# B&R Automation Studio project VisionSample (part 4)

#### Main.st - Init, cyclic, exit code
```iecst
// --------------------------------------------------------------------------------------------------------------------
// Vision image upload task. This task stores the camera image on the file device media
// Version 2.0
// --------------------------------------------------------------------------------------------------------------------
PROGRAM _INIT
	gVisionImage.CFG.FileDevice 	:= 'VisionFileDevice';		// File device name where the images are stored
	gVisionImage.CFG.DirName		:= 'Vision';				// Directory used for images

	gVisionImage.CMD.CreateDir	:= TRUE;
	gVisionImage.DAT.ImageSelected	:= '';

	brsmemcpy(ADR(b64key), ADR('ABCDEFGHIJKLMNOPQRSTUVWXYZabcdefghijklmnopqrstuvwxyz0123456789+/'), SIZEOF(b64key));

	// Create memory for uploading and transforming image
	// Size: a 5MP picture in bmp format has less than 6.000.000 Bytes. A SVG with bas64 conversion maximum the 4/3 size.
	MemUploadSize		:= 6000000;
	MemSvgHeaderSize	:= 2000;
	MemSvgCrosshSize	:= 18000;
	MemSvgSize			:= MemUploadSize * 4 / 3 + MemSvgHeaderSize + MemSvgCrosshSize;
	AsMemPartCreate_0.enable	:= TRUE;
	AsMemPartCreate_0.len		:= MemUploadSize + MemSvgSize + MemSvgCrosshSize + 1000; // 1000 Bytes for AsMemPart stuff/header
	AsMemPartCreate_0();

	IF AsMemPartCreate_0.status = 0 THEN
		AsMemPartAllocClear_0.enable	:= TRUE;
		AsMemPartAllocClear_0.ident		:= AsMemPartCreate_0.ident;
		AsMemPartAllocClear_0.len		:= MemUploadSize;
		AsMemPartAllocClear_0();
		IF AsMemPartAllocClear_0.status = 0 THEN
			MemUpload := AsMemPartAllocClear_0.mem;
		END_IF
		AsMemPartAllocClear_0.len		:= MemSvgSize;
		AsMemPartAllocClear_0();
		IF AsMemPartAllocClear_0.status = 0 THEN
			MemSvg := AsMemPartAllocClear_0.mem;
		END_IF
		AsMemPartAllocClear_0.len		:= MemSvgCrosshSize;
		AsMemPartAllocClear_0();
		IF AsMemPartAllocClear_0.status = 0 THEN
			MemSvgCrossh := AsMemPartAllocClear_0.mem;
		END_IF
	END_IF
	ACTION_InitTexts;
END_PROGRAM

// -----------------------------------------------------------------------------------------------------------
// Cyclic part
// -----------------------------------------------------------------------------------------------------------
PROGRAM _CYCLIC

	// -----------------------------------------------------------------------------------------------------------
	// State machine for uploading the image
	// -----------------------------------------------------------------------------------------------------------
	CASE Step OF
		// -----------------------------------------------------------------------------------------------------------
		// Wait for new upload command
		VISTEP_WAIT:
			gVisionImage.DAT.Status := 0;

			// -----------------------------------------------------------------------------------------------------------
			// Create the internal directory VisionImageArchive
			IF gVisionImage.CMD.CreateDir THEN
				gVisionImage.DAT.Status := 65535;
				Step := VISTEP_CREATE_DIR;

			// -----------------------------------------------------------------------------------------------------------
			// Delete image directory
			ELSIF gVisionImage.CMD.DeleteDir THEN
				gVisionImage.DAT.Status := 65535;
				Step := VISTEP_DELETE_DIR;

			// -----------------------------------------------------------------------------------------------------------
			// Refresh image data from file device
			ELSIF gVisionImage.CMD.Refresh THEN
				gVisionImage.DAT.Status := 65535;
				Step := VISTEP_READ_DIR1;

			// -----------------------------------------------------------------------------------------------------------
			// Delete image data from file device
			ELSIF gVisionImage.CMD.DeleteImage THEN
				IF brsstrlen(ADR(gVisionImage.DAT.ImageSelected)) > 0 THEN
					brsstrcpy(ADR(FileNamePict), ADR(gVisionImage.CFG.DirName));
					brsstrcat(ADR(FileNamePict), ADR('/'));
					brsstrcat(ADR(FileNamePict), ADR(gVisionImage.DAT.ImageSelected));
					gVisionImage.DAT.Status := 65535;
					Step := VISTEP_DELETE_IMAGE;
				ELSE
					gVisionImage.CMD.DeleteImage := FALSE;
				END_IF

				// -----------------------------------------------------------------------------------------------------------
				// Save image from camera
			ELSIF gVisionImage.CMD.GetImage THEN
				FileNamePict := gVisionImage.CFG.DirName;
				brsstrcat(ADR(FileNamePict), ADR('/last_image.bmp'));

				ViBaseGetImage_0.Execute := FALSE;
				ViBaseGetImage_0();

				gVisionImage.DAT.Status		:= 65535;
				Step						:= VISTEP_DELETE_IMAGE;

				// -----------------------------------------------------------------------------------------------------------
				// Save image from camera
			ELSIF gVisionImage.CMD.SaveImage THEN
				// Generate file name if not provided
				IF gVisionImage.CFG.FileName = '' THEN
					// Generate new file name
					DTGetTime_0.enable := 1;
					DTGetTime_0();
					DT_TO_DTStructure(DTGetTime_0.DT1, ADR(DTStructure_0));
					FileNamePict := gVisionImage.CFG.DirName;
					brsstrcat(ADR(FileNamePict), ADR('/'));
					tmpStr1 := UINT_TO_STRING(DTStructure_0.year);
					brsstrcat(ADR(FileNamePict), ADR(tmpStr1));
					brsstrcat(ADR(FileNamePict), ADR('_'));
					tmpStr1 := USINT_TO_STRING(DTStructure_0.month);
					IF(DTStructure_0.month < 10) THEN
						brsstrcat(ADR(FileNamePict), ADR('0'));
					END_IF
					brsstrcat(ADR(FileNamePict), ADR(tmpStr1));
					brsstrcat(ADR(FileNamePict), ADR('_'));
					tmpStr1 := USINT_TO_STRING(DTStructure_0.day);
					IF(DTStructure_0.day < 10) THEN
						brsstrcat(ADR(FileNamePict), ADR('0'));
					END_IF
					brsstrcat(ADR(FileNamePict), ADR(tmpStr1));
					brsstrcat(ADR(FileNamePict), ADR('_'));
					tmpStr1 := USINT_TO_STRING(DTStructure_0.hour);
					IF(DTStructure_0.hour < 10) THEN
						brsstrcat(ADR(FileNamePict), ADR('0'));
					END_IF
					brsstrcat(ADR(FileNamePict), ADR(tmpStr1));
					brsstrcat(ADR(FileNamePict), ADR('_'));
					tmpStr1 := USINT_TO_STRING(DTStructure_0.minute);
					IF(DTStructure_0.minute < 10) THEN
						brsstrcat(ADR(FileNamePict), ADR('0'));
					END_IF
					brsstrcat(ADR(FileNamePict), ADR(tmpStr1));
					brsstrcat(ADR(FileNamePict), ADR('_'));
					tmpStr1 := USINT_TO_STRING(DTStructure_0.second);
					IF(DTStructure_0.second < 10) THEN
						brsstrcat(ADR(FileNamePict), ADR('0'));
					END_IF
					brsstrcat(ADR(FileNamePict), ADR(tmpStr1));
				ELSE
					FileNamePict := gVisionImage.CFG.FileName;
				END_IF

				brsstrcpy(ADR(FileNameSvg), ADR(FileNamePict));
				brsstrcat(ADR(FileNameSvg), ADR('.svg'));
				brsstrcat(ADR(FileNamePict), ADR('.bmp'));

				ViBaseGetImage_0.Execute := FALSE;
				ViBaseGetImage_0();

				gVisionImage.DAT.Status		:= 65535;
				Step						:= VISTEP_DELETE_IMAGE;

			// -----------------------------------------------------------------------------------------------------------
			// Reset error
			ELSIF gVisionImage.CMD.ResetError THEN
				gVisionImage.CMD.ResetError := FALSE;
			END_IF

			// -----------------------------------------------------------------------------------------------------------
			// Load new image into window
			IF visImageSelectedOld <> gVisionImage.DAT.ImageSelected AND dir_entry > 0 THEN
				brsmemset(ADR(gVisionImage.DAT.ImagePath), 0, SIZEOF(gVisionImage.DAT.ImagePath));
				brsmemset(ADR(tmpStr1), 0, SIZEOF(tmpStr1));
				gVisionImage.DAT.ImagePath := '/FileDevice:';
				brsstrcat(ADR(gVisionImage.DAT.ImagePath), ADR(gVisionImage.CFG.FileDevice));
				brsstrcat(ADR(gVisionImage.DAT.ImagePath), ADR('/'));
				brsstrcat(ADR(gVisionImage.DAT.ImagePath), ADR(gVisionImage.CFG.DirName));
				brsstrcat(ADR(gVisionImage.DAT.ImagePath), ADR('/'));
				brsstrcat(ADR(gVisionImage.DAT.ImagePath), ADR(gVisionImage.DAT.ImageSelected));
			END_IF
			visImageSelectedOld := gVisionImage.DAT.ImageSelected;

		// -----------------------------------------------------------------------------------------------------------
		// Create directory on User-Partition, if not exists
		// -----------------------------------------------------------------------------------------------------------
		VISTEP_CREATE_DIR:
			DirCreate_0.enable	:= TRUE;
			DirCreate_0.pDevice	:= ADR(gVisionImage.CFG.FileDevice);
			DirCreate_0.pName	:= ADR(gVisionImage.CFG.DirName);
			DirCreate_0();

			IF DirCreate_0.status = 0 OR DirCreate_0.status = fiERR_DIR_ALREADY_EXIST THEN
				Step := VISTEP_READ_DIR1;
			ELSIF DirCreate_0.status <> 65535 THEN
				gVisionImage.DAT.Status := DirCreate_0.status;
				Step := VISTEP_ERR;
			END_IF

		// -----------------------------------------------------------------------------------------------------------
		// Delete directory on User-Partition
		// -----------------------------------------------------------------------------------------------------------
		VISTEP_DELETE_DIR:
			DirDeleteEx_0.enable	:= TRUE;
			DirDeleteEx_0.pDevice	:= ADR(gVisionImage.CFG.FileDevice);
			DirDeleteEx_0.pName		:= ADR(gVisionImage.CFG.DirName);
			DirDeleteEx_0();

			IF DirDeleteEx_0.status = 0 THEN
				Step := VISTEP_CREATE_DIR;
			ELSIF DirDeleteEx_0.status <> 65535 THEN
				gVisionImage.DAT.Status := DirDeleteEx_0.status;
				Step := VISTEP_ERR;
			END_IF

		// -----------------------------------------------------------------------------------------------------------
		// Read all existing image names from directory
		// -----------------------------------------------------------------------------------------------------------
		VISTEP_READ_DIR1:
			// Clear all memory
			brsmemset(ADR(gVisionImage.DAT.ImagesList), 0, SIZEOF(gVisionImage.DAT.ImagesList));
			brsmemset(ADR(gVisionImage.DAT.ImageSelected), 0, SIZEOF(gVisionImage.DAT.ImageSelected));
			visImageSelectedOld := '';
			gVisionImage.DAT.ImageSelected	:= '';
			dir_entry			:= 0;
			idx					:= 0;
			file_newest			:= '';
			file_oldest			:= '';
			date_newest			:= UDINT_TO_DT(0);
			date_oldest			:= DT#2100-06-06-12:00:00;
			cmdDeleteOldest		:= FALSE;
			Step := VISTEP_READ_DIR2;

		// -----------------------------------------------------------------------------------------------------------
		// Proceed with next entry
		// -----------------------------------------------------------------------------------------------------------
		VISTEP_READ_DIR2:
			DirRead_0.enable 	:= 1;
			DirRead_0.pDevice 	:= ADR(gVisionImage.CFG.FileDevice);
			DirRead_0.pPath		:= ADR(gVisionImage.CFG.DirName);
			DirRead_0.entry 	:= idx;
			DirRead_0.option 	:= fiFILE;
			DirRead_0.pData 	:= ADR(dir_data);
			DirRead_0.data_len 	:= SIZEOF(dir_data);
			DirRead_0();

			IF DirRead_0.status = 0 THEN
				// Make sure file is an image and we have space to store them
				IF  brsstrcmp(ADR(dir_data.Filename) + brsstrlen(ADR(dir_data.Filename)) - 4, ADR('.bmp')) = 0 OR
					brsstrcmp(ADR(dir_data.Filename) + brsstrlen(ADR(dir_data.Filename)) - 4, ADR('.jpg')) = 0 OR
					brsstrcmp(ADR(dir_data.Filename) + brsstrlen(ADR(dir_data.Filename)) - 4, ADR('.svg')) = 0 THEN
					// Find newest and oldest file
					IF dir_data.Date > date_newest THEN
						brsstrcpy(ADR(file_newest), ADR(dir_data.Filename));
						date_newest := dir_data.Date;
					END_IF
					IF dir_data.Date < date_oldest THEN
						brsstrcpy(ADR(file_oldest), ADR(dir_data.Filename));
						date_oldest := dir_data.Date;
					END_IF
					IF dir_entry <= SIZEOF(gVisionImage.DAT.ImagesList)/SIZEOF(gVisionImage.DAT.ImagesList[0]) - 1 THEN
						// Create list box data
						gVisionImage.DAT.ImagesList[dir_entry] := '{"value":"';
						brsstrcat(ADR(gVisionImage.DAT.ImagesList[dir_entry]), ADR(dir_data.Filename));
						brsstrcat(ADR(gVisionImage.DAT.ImagesList[dir_entry]), ADR('","text":"'));
						brsstrcat(ADR(gVisionImage.DAT.ImagesList[dir_entry]), ADR(dir_data.Filename));
						brsstrcat(ADR(gVisionImage.DAT.ImagesList[dir_entry]), ADR('"}'));
						dir_entry := dir_entry + 1;
					ELSE
						cmdDeleteOldest := TRUE;
					END_IF
				END_IF
				idx := idx + 1;
			ELSIF DirRead_0.status = fiERR_NO_MORE_ENTRIES THEN
				IF cmdDeleteOldest THEN
					brsstrcpy(ADR(tmpStr1), ADR(gVisionImage.CFG.DirName));
					brsstrcat(ADR(tmpStr1), ADR('/'));
					brsstrcat(ADR(tmpStr1), ADR(file_oldest));
					Step := VISTEP_DELETE_IMAGE;
				ELSE
					TON_VisPause(IN := FALSE);
					Step := VISTEP_READ_DIR3;
				END_IF
			ELSIF DirRead_0.status <> 65535 THEN
				gVisionImage.DAT.Status := DirRead_0.status;
				Step := VISTEP_ERR;
			END_IF

		// -----------------------------------------------------------------------------------------------------------
		// Wait for vis before setting last file
		// -----------------------------------------------------------------------------------------------------------
		VISTEP_READ_DIR3:
			TON_VisPause.IN := TRUE;
			TON_VisPause.PT := T#250ms;
			TON_VisPause();

			IF TON_VisPause.Q THEN
				brsstrcpy(ADR(gVisionImage.DAT.ImageSelected), ADR(file_newest));
				brsmemset(ADR(gVisionImage.CMD), 0, SIZEOF(gVisionImage.CMD));
				Step := VISTEP_WAIT;
			END_IF

		// -----------------------------------------------------------------------------------------------------------
		// Delete Image
		// -----------------------------------------------------------------------------------------------------------
		VISTEP_DELETE_IMAGE:
			cmdDeleteOldest			:= FALSE;
			FileDelete_0.enable 	:= 1;
			FileDelete_0.pDevice	:= ADR(gVisionImage.CFG.FileDevice);
			FileDelete_0.pName 		:= ADR(FileNamePict);
			FileDelete_0();

			IF (FileDelete_0.status = 0 OR FileDelete_0.status = fiERR_FILE_NOT_FOUND) AND (gVisionImage.CMD.GetImage OR gVisionImage.CMD.SaveImage) THEN
				Step := VISTEP_REQUEST;
			ELSIF FileDelete_0.status = 0 THEN
				Step := VISTEP_READ_DIR1;
			ELSIF FileDelete_0.status <> 65535 THEN
				gVisionImage.DAT.Status := FileDelete_0.status;
				Step := VISTEP_ERR;
			END_IF

		// -----------------------------------------------------------------------------------------------------------
		// Get new image
		// -----------------------------------------------------------------------------------------------------------
		VISTEP_REQUEST:
			ViBaseGetImage_0.MpLink := ADR(gVisionImage.CFG.ComponentLink);
			ViBaseGetImage_0.Execute := TRUE;
			ViBaseGetImage_0.Type :=  viBASE_IMAGE_TYPE_BMP;
			//ViBaseGetImage_0.QualityLevel := ;
			ViBaseGetImage_0.Timeout := T#10s;
			ViBaseGetImage_0.Buffer := MemUpload;
			ViBaseGetImage_0.BufferSize := MemUploadSize;
			ViBaseGetImage_0();

			IF ViBaseGetImage_0.Busy = 0 THEN
				IF ViBaseGetImage_0.StatusID = 0 THEN
					Step := VISTEP_SAVE1;
				ELSIF ViBaseGetImage_0.StatusID <> ERR_FUB_BUSY THEN
					gVisionImage.DAT.Status := ViBaseGetImage_0.StatusID;
					Step := VISTEP_ERR;
				END_IF
			END_IF

		// -----------------------------------------------------------------------------------------------------------
		// Save image
		// -----------------------------------------------------------------------------------------------------------
		VISTEP_SAVE1:
			FileCreate_0.enable		:= TRUE;
			FileCreate_0.pDevice	:= ADR(gVisionImage.CFG.FileDevice);
			FileCreate_0.pFile		:= ADR(FileNamePict);
			FileCreate_0();

			IF FileCreate_0.status = 0 THEN
				Step := VISTEP_SAVE2;
			ELSIF FileCreate_0.status <> ERR_FUB_BUSY THEN
				gVisionImage.DAT.Status := FileCreate_0.status;
				Step := VISTEP_ERR;
			END_IF

		VISTEP_SAVE2:
			FileWrite_0.enable		:= TRUE;
			FileWrite_0.ident		:= FileCreate_0.ident;
			FileWrite_0.offset		:= 0;
			FileWrite_0.pSrc		:= MemUpload;
			FileWrite_0.len			:= ViBaseGetImage_0.BufferLen;
			FileWrite_0();

			IF FileWrite_0.status = 0 THEN
				Step := VISTEP_SAVE3;
			ELSIF FileWrite_0.status <> ERR_FUB_BUSY THEN
				gVisionImage.DAT.Status := FileWrite_0.status;
				Step := VISTEP_ERR;
			END_IF

		VISTEP_SAVE3:
			FileClose_0.enable		:= TRUE;
			FileClose_0.ident		:= FileCreate_0.ident;
			FileClose_0();

			IF FileClose_0.status = 0 THEN
				image_idx := image_idx + 1;
				brsitoa(image_idx, ADR(tmpStr1));
				gVisionImage.DAT.ImageLast := '/FileDevice:';
				brsstrcat(ADR(gVisionImage.DAT.ImageLast), ADR(gVisionImage.CFG.FileDevice));
				brsstrcat(ADR(gVisionImage.DAT.ImageLast), ADR('/'));
				brsstrcat(ADR(gVisionImage.DAT.ImageLast), ADR(gVisionImage.CFG.DirName));
				brsstrcat(ADR(gVisionImage.DAT.ImageLast), ADR('/last_image.bmp?'));
				brsstrcat(ADR(gVisionImage.DAT.ImageLast), ADR(tmpStr1));

				IF gVisionImage.CMD.SaveImage THEN
					Step := VISTEP_SVG_PREPARE;
				ELSE
					gVisionImage.CMD.GetImage := FALSE;
					Step := VISTEP_WAIT;
				END_IF
			ELSIF FileClose_0.status <> ERR_FUB_BUSY THEN
				gVisionImage.DAT.Status := FileClose_0.status;
				Step := VISTEP_ERR;
			END_IF

		// -----------------------------------------------------------------------------------------------------------
		// Create SVG file with image and crosshair/texts
		// -----------------------------------------------------------------------------------------------------------
		VISTEP_SVG_PREPARE:
			b64neededOutput	:= (ViBaseGetImage_0.BufferLen/3)*4 + BOOL_TO_UDINT(UDINT_TO_BOOL(ViBaseGetImage_0.BufferLen MOD 3))*4;
			IF b64neededOutput < MemSvgSize - MemSvgHeaderSize - MemSvgCrosshSize THEN
				brsmemset(MemSvg, 0, MemSvgSize); // clear complete memory
				// Prepare the svg header up to the base64 picture data
				brsstrcpy(MemSvg, ADR(SvgTexts.Header1));
				brsstrcat(MemSvg, ADR(FileNameSvg));
				brsstrcat(MemSvg, ADR(SvgTexts.Header2));
				brsstrcat(MemSvg, ADR('bmp'));
				brsstrcat(MemSvg, ADR(SvgTexts.Header3));
				Step := VISTEP_SVG_BAS64_1;
			ELSE
				gVisionImage.DAT.Status := ERR_BUFF_TOO_SMALL;
				Step := VISTEP_ERR;
			END_IF

		// -----------------------------------------------------------------------------------------------------------
		// Code picture data with Base64 to embedd the picture into a svg file
		VISTEP_SVG_BAS64_1:
			b64AdrInBuffer	:= MemUpload; 						// Original bmp or jpg picture
			b64AdrOutBuffer	:= MemSvg + brsstrlen(MemSvg); 		// Write to the end of the actual svg data
			b64actposIN		:= b64AdrInBuffer;
			b64actposOUT	:= b64AdrOutBuffer;
			Step := VISTEP_SVG_BAS64_2;

		VISTEP_SVG_BAS64_2:
			FOR i := 0 TO CONVERT_CYCLES DO
				IF b64actposIN < b64AdrInBuffer + ViBaseGetImage_0.BufferLen THEN
					b64blockLen := UDINT_TO_USINT(LIMIT(0, b64AdrInBuffer + ViBaseGetImage_0.BufferLen - b64actposIN, 3));
					b64in ACCESS b64actposIN;
					b64out ACCESS b64actposOUT;
					b64out[0]		:= b64key[ SHR(b64in[0],2) ];
					IF b64blockLen = 1 THEN
						b64out[1]	:= b64key[ SHL((b64in[0] AND 16#03),4)];
						b64out[2]	:= 61;
						b64out[3]	:= 61;
					ELSIF b64blockLen = 2 THEN
						b64out[1]	:= b64key[ SHL((b64in[0] AND 16#03),4) OR SHR(b64in[1],4) ];
						b64out[2]	:= b64key[ SHL((b64in[1] AND 16#0F),2)];
						b64out[3]	:= 61;
					ELSIF b64blockLen = 3 THEN
						b64out[1]	:= b64key[ SHL((b64in[0] AND 16#03),4) OR SHR(b64in[1],4) ];
						b64out[2]	:= b64key[ SHL((b64in[1] AND 16#0F),2) OR SHR(b64in[2],6) ];
						b64out[3]	:= b64key[ b64in[2] AND 16#3F ];
					END_IF
					b64actposIN		:= b64actposIN + 3;
					b64actposOUT	:= b64actposOUT + 4;
				ELSE
					Step := VISTEP_SVG_CROSSH;
					EXIT;
				END_IF

			END_FOR

		// -----------------------------------------------------------------------------------------------------------
		// Prepare the second part after base64 picture data
		VISTEP_SVG_CROSSH:
			brsmemset(MemSvgCrossh, 0, MemSvgCrosshSize);
			brsstrcat(MemSvgCrossh, ADR(SvgTexts.Header4));
			brsstrcat(MemSvgCrossh, ADR(SvgTexts.CrosshairDefinition));
			FOR i := 1 TO MAX_NUM_RESULTS DO
				IF gVisionImage.DAT.Crosshair[i].CrosshairX <> 0 AND gVisionImage.DAT.Crosshair[i].CrosshairY <> 0 THEN
					brsstrcat(MemSvgCrossh, ADR(SvgTexts.Crosshair1));
					brsitoa(REAL_TO_DINT(gVisionImage.DAT.Crosshair[i].CrosshairX), ADR(tmpStr1));
					brsstrcat(MemSvgCrossh, ADR(tmpStr1));
					brsstrcat(MemSvgCrossh, ADR(','));
					brsitoa(REAL_TO_DINT(gVisionImage.DAT.Crosshair[i].CrosshairY), ADR(tmpStr1));
					brsstrcat(MemSvgCrossh, ADR(tmpStr1));
					brsstrcat(MemSvgCrossh, ADR(') rotate('));
					brsitoa(REAL_TO_DINT(gVisionImage.DAT.Crosshair[i].CrosshairRotate), ADR(tmpStr1));
					brsstrcat(MemSvgCrossh, ADR(tmpStr1));
					brsstrcat(MemSvgCrossh, ADR(',40,40)"/>'));
				END_IF
			END_FOR
			FOR i := 1 TO MAX_NUM_RESULTS DO
				IF gVisionImage.DAT.Crosshair[i].CrosshairX <> 0 AND gVisionImage.DAT.Crosshair[i].CrosshairY <> 0 THEN
					brsstrcat(MemSvgCrossh, ADR('$r$n$t'));
					brsstrcat(MemSvgCrossh, ADR(gVisionImage.DAT.Crosshair[i].Text));
				END_IF
			END_FOR
			brsstrcat(MemSvgCrossh, ADR(SvgTexts.SvgClose));
			Step := VISTEP_SVG_CONCAT;

		VISTEP_SVG_CONCAT:
			brsstrcat(MemSvg, MemSvgCrossh);
			Step := VISTEP_SVG_SAVE1;

		// -----------------------------------------------------------------------------------------------------------
		// Save SVG file
		// -----------------------------------------------------------------------------------------------------------
		VISTEP_SVG_SAVE1:
			FileCreate_0.enable		:= TRUE;
			FileCreate_0.pDevice	:= ADR(gVisionImage.CFG.FileDevice);
			FileCreate_0.pFile		:= ADR(FileNameSvg);
			FileCreate_0();

			IF FileCreate_0.status = 0 THEN
				Step := VISTEP_SVG_SAVE2;
			ELSIF FileCreate_0.status <> ERR_FUB_BUSY THEN
				gVisionImage.DAT.Status := FileCreate_0.status;
				Step := VISTEP_ERR;
			END_IF

		VISTEP_SVG_SAVE2:
			FileWrite_0.enable		:= TRUE;
			FileWrite_0.ident		:= FileCreate_0.ident;
			FileWrite_0.offset		:= 0;
			FileWrite_0.pSrc		:= MemSvg;
			FileWrite_0.len			:= brsstrlen(MemSvg);
			FileWrite_0();

			IF FileWrite_0.status = 0 THEN
				Step := VISTEP_SVG_SAVE3;
			ELSIF FileWrite_0.status <> ERR_FUB_BUSY THEN
				gVisionImage.DAT.Status := FileWrite_0.status;
				Step := VISTEP_ERR;
			END_IF

		VISTEP_SVG_SAVE3:
			FileClose_0.enable		:= TRUE;
			FileClose_0.ident		:= FileCreate_0.ident;
			FileClose_0();

			IF FileClose_0.status = 0 THEN
				Step := VISTEP_READ_DIR1;
			ELSIF FileClose_0.status <> ERR_FUB_BUSY THEN
				gVisionImage.DAT.Status := FileClose_0.status;
				Step := VISTEP_ERR;
			END_IF

		// -----------------------------------------------------------------------------------------------------------
		// Error state
		// -----------------------------------------------------------------------------------------------------------
		VISTEP_ERR:
			// Reset all commands and wait or ack
			ViBaseGetImage_0.Execute	:= TRUE;
			ViBaseGetImage_0();

			IF gVisionImage.CMD.ResetError THEN
				gVisionImage.CMD.ResetError := FALSE;
				Step := VISTEP_WAIT;
			END_IF
			brsmemset(ADR(gVisionImage.CMD), 0, SIZEOF(gVisionImage.CMD));
	END_CASE

END_PROGRAM
```

#### Types.typ - Local data types
```iecst
TYPE
	VIStep_Enum :
		(
		VISTEP_WAIT,
		VISTEP_GEN_CROSSHAIR,
		VISTEP_CREATE_DIR,
		VISTEP_DELETE_DIR,
		VISTEP_READ_DIR1,
		VISTEP_READ_DIR2,
		VISTEP_READ_DIR3,
		VISTEP_DELETE_IMAGE,
		VISTEP_REQUEST1,
		VISTEP_REQUEST2,
		VISTEP_REQUEST3,
		VISTEP_SAVE1,
		VISTEP_SAVE2,
		VISTEP_SAVE3,
		VISTEP_SVG_CROSSH,
		VISTEP_SVG_CONCAT,
		VISTEP_ERR
		);
	SvgTexts_Type : 	STRUCT
		Header1 : STRING[500];
		Header2 : STRING[500];
		Header3 : STRING[500];
		Header4 : STRING[500];
		CrosshairDefinition : STRING[1000];
		Crosshair1 : STRING[500];
		SvgClose : STRING[50];
	END_STRUCT;
	DiagTime_Type : 	STRUCT
		Refresh : TIME;
		BeginSaveBMPJPG : TIME;
		EndSaveBMPJPG : TIME;
		BeginSVG : TIME;
		BeginSVGSave : TIME;
		EndSVGSave : TIME;
	END_STRUCT;
END_TYPE
```

#### Variables.var - Local variables
```iecst
VAR
	Step : VIStep_Enum;
	tmpStr1 : STRING[80];
	idx : UINT;
END_VAR
(**)
(*Filehandling*)
VAR
	DirCreate_0 : DirCreate;
	DirDeleteEx_0 : DirDeleteEx;
	FileNamePict : STRING[80];
	FileNameSvg : STRING[80];
	FileCreate_0 : FileCreate;
	FileDelete_0 : FileDelete;
	FileWrite_0 : FileWrite;
	FileClose_0 : FileClose;
	DirRead_0 : DirRead;
	dir_data : fiDIR_READ_DATA;
	dir_entry : UINT;
	file_newest : STRING[80];
	file_oldest : STRING[80];
	date_newest : DATE_AND_TIME;
	date_oldest : DATE_AND_TIME;
	cmdDeleteOldest : BOOL;
	image_idx : UINT;
	DTGetTime_0 : DTGetTime;
	DTStructure_0 : DTStructure;
	TON_VisPause : TON;
END_VAR
(**)
(*mappView connected variables*)
VAR
	visImageSelectedOld : STRING[80];
END_VAR
(**)
(*Create memory*)
VAR
	AsMemPartCreate_0 : AsMemPartCreate;
	AsMemPartAllocClear_0 : AsMemPartAllocClear;
	MemUpload : UDINT;
	MemUploadSize : UDINT;
	MemSvg : UDINT;
	MemSvgSize : UDINT;
	MemSvgHeaderSize : UDINT;
	MemSvgCrossh : UDINT;
	MemSvgCrosshSize : UDINT;
END_VAR
(**)
VAR
	ViBaseGetImage_0 : ViBaseGetImage;
END_VAR
(**)
(*Bas64*)
VAR
	b64AdrInBuffer : UDINT;
	b64AdrOutBuffer : UDINT;
	b64neededOutput : UDINT;
	b64key : ARRAY[0..63] OF USINT;
	b64actposIN : UDINT;
	b64actposOUT : UDINT;
	b64in : REFERENCE TO ARRAY[0..2] OF USINT;
	b64out : REFERENCE TO ARRAY[0..3] OF USINT;
	b64blockLen : USINT;
	SvgTexts : SvgTexts_Type;
	i : UDINT;
END_VAR
(**)
(*Constants*)
VAR
	ERR_BUFF_TOO_SMALL : UINT := 50001;
END_VAR
```

#### LocalFunctions.fun - not listed in the package file held
```iecst
FUNCTION_BLOCK ViDownloadImage (* *) (*$GROUP=User,$CAT=User,$GROUPICON=User.png,$CATICON=User.png*)
	VAR_INPUT
		Enable : BOOL;
		FileDevice : STRING[80];
		FileName : STRING[80];
		ImgName : STRING[80];
		visDownloadFileUrl : REFERENCE TO STRING[200];
	END_VAR
	VAR_OUTPUT
		Status : UINT;
	END_VAR
	VAR
		Step : INT;
		AsMemPartCreate_0 : AsMemPartCreate;
		AsMemPartAllocClear_0 : AsMemPartAllocClear;
		MemSvgAdr : UDINT;
		MemSvgSize : UDINT;
		FileOpen_0 : FileOpen;
		FileRead_0 : FileRead;
		FileClose_0 : FileClose;
		TON_Timeout : TON;
		httpService_Download : httpService;
		response_header : httpResponseHeader_t;
		response_header_data : STRING[300];
	END_VAR
END_FUNCTION_BLOCK

FUNCTION_BLOCK ViRefreshImageList
	VAR_INPUT
		Enable : BOOL;
		VisionImage : REFERENCE TO typVisionImage;
		ImageList : REFERENCE TO ARRAY[0..19] OF STRING[80];
		visSelectedImage : REFERENCE TO STRING[80];
	END_VAR
	VAR_OUTPUT
		Status : UINT;
		DirEntries : UINT;
	END_VAR
	VAR
		Step : INT;
		visSelectedImageOld : STRING[80];
		idx : UINT;
		file_newest : STRING[80];
		file_oldest : STRING[80];
		date_newest : DATE_AND_TIME;
		date_oldest : DATE_AND_TIME;
		cmdDeleteOldest : BOOL;
		DirRead_0 : DirRead;
		FileDelete_0 : FileDelete;
		dir_data : fiDIR_READ_DATA;
		DeleteFileName : STRING[80];
		TON_VisPause : TON;
	END_VAR
END_FUNCTION_BLOCK

FUNCTION_BLOCK ViSaveImgOnPlc
	VAR_INPUT
		Enable : BOOL;
		CFG : typVisionImageConfig;
		PowerlinkNode : USINT;
		CrossHairInfo : REFERENCE TO ARRAY[0..MAX_NUM_RESULTS] OF typCrossHairInfo;
	END_VAR
	VAR_OUTPUT
		Status : UINT;
	END_VAR
	VAR
		Step : INT;
		AsMemPartCreate_0 : AsMemPartCreate;
		AsMemPartAllocClear_0 : AsMemPartAllocClear;
		MemInfo : MemInfoSave_Type;
		DiagStartTime : TIME;
		DiagTime : DiagTime_Type;
		DTGetTime_0 : DTGetTime;
		DTStructure_0 : DTStructure;
		FileNameImg : STRING[80];
		FileNameSvg : STRING[80];
		URI : STRING[80];
		Host : STRING[80];
		httpClient_0 : httpClient;
		httpClientErrorStatus : UINT;
		RequestHeader : httpRequestHeader_t;
		TON_ReloadTimeout : TON;
		UploadedImgSize : UDINT;
		FileCreate_0 : FileCreate;
		FileWrite_0 : FileWrite;
		FileClose_0 : FileClose;
		b64AdrInBuffer : UDINT;
		b64AdrOutBuffer : UDINT;
		b64neededOutput : UDINT;
		b64key : ARRAY[0..63] OF USINT;
		b64actposIN : UDINT;
		b64actposOUT : UDINT;
		b64in : REFERENCE TO ARRAY[0..2] OF USINT;
		b64out : REFERENCE TO ARRAY[0..3] OF USINT;
		b64blockLen : UINT;
		FirstElement : BOOL;
		SvgTexts : SvgTexts_Type;
		tmpStr1 : STRING[80];
		i : UDINT;
	END_VAR
END_FUNCTION_BLOCK

FUNCTION_BLOCK ViDrawCrosshair
	VAR_INPUT
		SelectedSensor : UINT;
		CmdRefreshCrosshair : BOOL;
		VisionSensor : REFERENCE TO typVisionMain;
		CodeTypes : REFERENCE TO ARRAY[0..MAX_NUM_CODETYPES] OF STRING[80];
		VisionDisabled : BOOL;
		TextAlignment : BOOL; (*0: left, 1: right*)
		ImageRotation_deg : UINT;
		visCrossHair : REFERENCE TO typCrossHair;
	END_VAR
	VAR_OUTPUT
		CrossHairInfo : ARRAY[0..MAX_NUM_RESULTS] OF typCrossHairInfo;
	END_VAR
	VAR
		idx : UINT;
		SelectedSensorOld : UINT;
		Blob : REFERENCE TO typBlobMain;
		CodeReader : REFERENCE TO typCodeReaderMain;
		Match : REFERENCE TO typMatchMain;
		MT : REFERENCE TO typMTMain;
		Pixel : REFERENCE TO typPixelMain;
		OCR : REFERENCE TO typOCRMain;
		DetailsNoOld : USINT;
		ShowCrosshairOld : BOOL;
		ImageRotation_degOld : UINT;
		TextAlignmentOld : BOOL;
		ResultModelNumber : USINT;
		ResultPositionX : REAL;
		ResultPositionY : REAL;
		ResultOrientation : REAL;
		CrosshSize : REAL;
		ScaleVertical : REAL;
		svgTrafo : STRING[200];
		svgContent : STRING[1000];
		tmpStr : STRING[100];
		blueTextPos : INT;
		MT_UseXY : BOOL;
	END_VAR
END_FUNCTION_BLOCK

FUNCTION_BLOCK ViCreateWebDirFile
	VAR_INPUT
		Enable : BOOL;
		FileDevUser : STRING[80];
		EthDevice : STRING[80];
		EthIP : STRING[80];
		visWebViewerPath : REFERENCE TO STRING[80];
	END_VAR
	VAR_OUTPUT
		Status : UINT;
		Done : BOOL;
	END_VAR
	VAR
		Step : INT;
		DirInfo_0 : DirInfo;
		DirCreate_0 : DirCreate;
		FileDelete_0 : FileDelete;
		FileCreate_0 : FileCreate;
		FileWrite_0 : FileWrite;
		FileClose_0 : FileClose;
		DevLink_0 : DevLink;
		FileCopy_0 : FileCopy;
		DevUnlink_0 : DevUnlink;
		FileDevSystem : STRING[80];
		FileDevSystemPara : STRING[80];
		DirNameWeb : STRING[80];
		FileNameVisImgHtml : STRING[80];
		FileNameEyeSystem : STRING[80];
		FileNameEyeUser : STRING[80];
		HtmlFileContent1 : STRING[1500];
		HtmlFileContent2 : STRING[2000];
		FileWriteData : STRING[3600];
	END_VAR
END_FUNCTION_BLOCK

FUNCTION_BLOCK ViShowImgOnVC4
	VAR_INPUT
		Enable : BOOL;
		RefreshImage : BOOL;
		CFG : typVisionImageConfig;
		PowerlinkNode : USINT;
		ImgWidthInVC4_px : UINT;
	END_VAR
	VAR_OUTPUT
		Status : UINT;
		HTMLStreamContent : STRING[600];
		RefreshDone : BOOL;
	END_VAR
	VAR
		Step : INT;
		AsMemPartCreate_0 : AsMemPartCreate;
		AsMemPartAllocClear_0 : AsMemPartAllocClear;
		MemInfo : MemInfoVC4_Type;
		FileNameBmp24Bit : STRING[80];
		FileNameBmp24BitDir : STRING[80];
		URI : STRING[80];
		Host : STRING[80];
		ImgHeight_px : UINT;
		httpClient_0 : httpClient;
		httpClientErrorStatus : UINT;
		RequestHeader : httpRequestHeader_t;
		TON_Timeout : TON;
		FileSizeIn8Bit : UDINT;
		FileDelete_0 : FileDelete;
		FileCreate_0 : FileCreate;
		FileWrite_0 : FileWrite;
		FileClose_0 : FileClose;
		Bmp8Bit : Bmp8Bit_Type;
		Bmp24Bit : Bmp24Bit_Type;
		BytesPerLine : DINT;
		PixelSourceAdr : UDINT;
		PixelDestAdr : UDINT;
		PixelSourceColor : REFERENCE TO USINT;
		PixelDestColor : REFERENCE TO PixelDestColor_Type;
		BytesRemaining : DINT;
		VC4HTML : ARRAY[0..3] OF STRING[300];
		tmpStr1 : STRING[30];
		i : UDINT;
	END_VAR
END_FUNCTION_BLOCK

FUNCTION CrosshairDetailsValue : BOOL
	VAR_INPUT
		strTarget : UDINT;
		strText : UDINT;
		fValue : REAL;
		TextAlignment : BOOL;
	END_VAR
	VAR
		tmpStr : STRING[80];
	END_VAR
END_FUNCTION

FUNCTION CrosshairDetailsText : BOOL
	VAR_INPUT
		strTarget : UDINT;
		strText : UDINT;
		adrText : UDINT;
		TextAlignment : BOOL;
	END_VAR
	VAR
		tmpStr : STRING[80];
	END_VAR
END_FUNCTION
```

#### Actions.st - not listed in the package file held
```iecst
ACTION ACTION_InitTexts:
SvgTexts.Header1 :=
'<?xml version="1.0" encoding="UTF-8"?>
<!DOCTYPE svg PUBLIC "-//W3C//DTD SVG 1.1//EN" "http://www.w3.org/Graphics/SVG/1.1/DTD/svg11.dtd">
<svg xmlns="http://www.w3.org/2000/svg" xml:space="preserve" width="1280px" height="1024px" shape-rendering="geometricPrecision" text-rendering="geometricPrecision" image-rendering="optimizeQuality" fill-rule="nonzero" clip-rule="evenodd" viewBox="0 0 1280 1024" xmlns:xlink="http://www.w3.org/1999/xlink">
	<title>';
SvgTexts.Header2 :=
'</title>
	<image
	xlink:href="data:image/';
SvgTexts.Header3 :=
';base64,';
SvgTexts.Header4 :=
'"
	width="1280"
	height="1024"
	id="LoadedPicture"
	x="0"
	y="0" />';
SvgTexts.CrosshairDefinition :=
'
	<defs>
		<symbol id="Fadenkreuz">
			<desc>Ein einfaches Fadenkreuz</desc>
			<g id="Crosshair">
			<path style="stroke:#ff0000;stroke-width:5" d="M 40,1 V 30 Z" id="up" />
			<path style="stroke:#ff0000;stroke-width:5" d="M 40,50 V 80 Z" id="down" />
			<path style="stroke:#ff0000;stroke-width:5" d="M 30,40 H 0 Z" id="left" />
			<path style="stroke:#ff0000;stroke-width:5" d="M 80,40 H 50 Z" id="right" />
			<circle style="fill:none;stroke:#ff0000;stroke-width:5" cx="40" cy="40" r="25" id="circle6" />
			</g>
		</symbol>
	</defs>';
SvgTexts.Crosshair1 :=
'
	<use xlink:href="#Fadenkreuz" transform="translate(';
SvgTexts.SvgClose :=
'
</svg>';

END_ACTION
```

#### CrosshairDetails.st - not listed in the package file held
```iecst
FUNCTION CrosshairDetailsValue
	IF NOT TextAlignment THEN // left
		tmpStr:= '<tspan text-anchor="start" class="text" x="10" dy="32">';
	ELSE // right
		tmpStr:= '<tspan text-anchor="end" class="text" x="1270" dy="32">';
	END_IF
	brsstrcat(strTarget, ADR(tmpStr));
	brsstrcat(strTarget, strText);
	brsftoa(fValue, ADR(tmpStr));
	brsstrcat(strTarget, ADR(tmpStr));
	brsstrcat(strTarget, ADR('</tspan> '));
	CrosshairDetailsValue := TRUE;
END_FUNCTION
FUNCTION CrosshairDetailsText
	IF NOT TextAlignment THEN // left
		tmpStr:= '<tspan text-anchor="start" class="text" x="10" dy="32">';
	ELSE // right
		tmpStr:= '<tspan text-anchor="end" class="text" x="1270" dy="32">';
	END_IF
	brsstrcat(strTarget, ADR(tmpStr));
	brsstrcat(strTarget, strText);
	brsstrcat(strTarget, adrText);
	brsstrcat(strTarget, ADR('</tspan> '));
	CrosshairDetailsText := TRUE;
END_FUNCTION
```

#### CrosshairDetailsText.st - not listed in the package file held
```iecst
FUNCTION CrosshairDetailsText
	tmpStr:= '<tspan class="text" x="10" dy="32">';
	brsstrcat(strTarget, ADR(tmpStr));
	brsstrcat(strTarget, strText);
	brsftoa(fValue, ADR(tmpStr));
	brsstrcat(strTarget, ADR(tmpStr));
	brsstrcat(strTarget, ADR('</tspan> '));
	CrosshairDetailsText := TRUE;
END_FUNCTION
```

#### LocalFunctions.st - not listed in the package file held
```iecst
FUNCTION_BLOCK ViDownloadImage
	visDownloadFileUrl ACCESS AdrVisDownloadFileUrl;
	IF NOT Enable THEN
		Status := ERR_FUB_ENABLE_FALSE;
	END_IF
	CASE Step OF
		0:
			Step := 10;
			Status := ERR_FUB_BUSY;
		10:
			FileOpen_0.enable	:= TRUE;
			FileOpen_0.pDevice 	:= ADR(FileDevice);
			FileOpen_0.pFile	:= ADR(FileName);
			FileOpen_0();
			IF FileOpen_0.status = 0 THEN
				IF FileOpen_0.filelen <= MemSize THEN // Make sure file fits into memory
					brsmemset(MemAdr, 0, MemSize);
					Step := 1;
				ELSE // File is too large
					Status := ERR_MEM_DOWNLOAD;
					Step := 0;
				END_IF
			ELSIF FileOpen_0.status <> ERR_FUB_BUSY THEN
				Status := FileOpen_0.status;
				Step := 0;
			END_IF
		1:
			FileRead_0.enable	:= TRUE;
			FileRead_0.ident	:= FileOpen_0.ident;
			FileRead_0.len		:= FileOpen_0.filelen;
			FileRead_0.pDest	:= MemAdr;
			FileRead_0();
			IF FileRead_0.status = 0 THEN
				Step := 2;
			ELSIF FileRead_0.status <> ERR_FUB_BUSY THEN
				Status := FileRead_0.status;
				Step := 0;
			END_IF
		2:
			FileClose_0.enable	:= TRUE;
			FileClose_0.ident	:= FileOpen_0.ident;
			FileClose_0();
			IF FileClose_0.status = 0 THEN
				TON_Timeout.IN := FALSE;
				TON_Timeout();
				Step := 3;
			ELSIF FileClose_0.status <> ERR_FUB_BUSY THEN
				Status := FileClose_0.status;
				Step := 0;
			END_IF
		3:
			httpService_Download.enable := FALSE;
			httpService_Download();
			Step := 4;
		4:
			// Create response header
			response_header_data :=  'Content-Type: application/octet-stream; Content-Transfer-Encoding: binary; Content-Disposition: attachment; filename="';
			brsstrcat(ADR(response_header_data), ADR(ImgName));
			brsstrcat(ADR(response_header_data), ADR('"'));
			// Pre-configure web service for download
			response_header.rawHeader.pData 	:= ADR(response_header_data);
			response_header.rawHeader.dataSize 	:= SIZEOF(response_header_data);
			response_header.rawHeader.dataLen 	:= brsstrlen(ADR(response_header_data));

			// ----------------------------------------------------------------------------------------
			// Start web service
			httpService_Download.enable 			:= TRUE;
			httpService_Download.option 			:= httpOPTION_HTTP_10 + httpOPTION_SERVICE_TYPE_NAME;
			httpService_Download.pResponseData 		:= MemAdr;
			httpService_Download.pResponseHeader	:= ADR(response_header);
			httpService_Download.pServiceName 		:= ADR(ImgName);
			httpService_Download.responseDataLen 	:= FileOpen_0.filelen;
			httpService_Download();

			// ----------------------------------------------------------------------------------------
			// Timeout if file is not pulled from browser
			TON_Timeout.IN := TRUE;
			TON_Timeout.PT := T#3s;
			TON_Timeout();
			IF TON_Timeout.Q THEN
				Status := ERR_TIMEOUT_DOWNLOAD;
				Step := 0;
			END_IF

			// ----------------------------------------------------------------------------------------
			// Set URL
			IF httpService_Download.status = ERR_FUB_BUSY AND visDownloadFileUrl = '' THEN
				brsstrcpy(ADR(visDownloadFileUrl), ADR(ImgName));
				// Start sending data
			ELSIF httpService_Download.status = 0 AND NOT httpService_Download.send AND visDownloadFileUrl <> '' THEN
				httpService_Download.send := TRUE;
			// Sending data finished
			ELSIF httpService_Download.send THEN
				Step := 5;
			// Error
			ELSIF httpService_Download.status <> ERR_FUB_BUSY AND httpService_Download.status <> 0 THEN
				Status := httpService_Download.status;
				Step := 0;
			END_IF
		// --------------------------------------------------------------------------------------------------------------------
		// Download file - web service
		// --------------------------------------------------------------------------------------------------------------------
		5:
			httpService_Download();
			TON_Timeout();
			IF TON_Timeout.Q THEN
				Status := ERR_TIMEOUT_DOWNLOAD;
				Step := 0;
			END_IF

			// ----------------------------------------------------------------------------------------
			// Start sending data
			IF httpService_Download.phase = httpPHASE_WAITING THEN
				//visDownloadFileUrl := '';
				httpService_Download.send := FALSE;
				Status := 0;
				Step := 0;
			ELSIF httpService_Download.status <> ERR_FUB_BUSY THEN
				Status := httpService_Download.status;
				Step := 0;
			END_IF
		100:
	END_CASE
END_FUNCTION_BLOCK
```

#### ViCreateWebDirFile.st - not listed in the package file held
```iecst
FUNCTION_BLOCK ViCreateWebDirFile
	IF NOT Enable THEN
		Status := ERR_FUB_ENABLE_FALSE;
		Step := 0;
		RETURN;
	END_IF
	CASE Step OF
		0:
			Status := ERR_FUB_BUSY;
			Done := FALSE;
			Step := 1;
		1: // Init
			ACTION_CreateHtmlFile;
			FileDevSystem		:= 'CF';
			FileDevSystemPara	:= '/DEVICE=C:/';
			DirNameWeb			:= 'web';
			FileNameVisImgHtml	:= 'web/VisionImg.html';
			FileNameEyeSystem	:= 'ADDONS/DATA/IAT_Data/wwwRoot/BRVisu/Media/VisionEye.png';
			FileNameEyeUser		:= 'web/VisionEye.png';
			Step := 2;
		2: // Check if web directory already exists
			DirInfo_0(enable := TRUE, pDevice := ADR(FileDevUser), pPath := ADR(DirNameWeb));
			IF DirInfo_0.status = ERR_OK THEN
				Step := 9;
			ELSIF DirInfo_0.status = fiERR_DIR_NOT_EXIST THEN
				Step := 3;
			ELSIF DirInfo_0.status <> ERR_FUB_BUSY THEN
				Status := DirInfo_0.status;
				Step := 0;
			END_IF
		3: // Create web directory if it does not exist
			DirCreate_0(enable := TRUE, pDevice := ADR(FileDevUser), pName := ADR(DirNameWeb));
			IF DirCreate_0.status = ERR_OK THEN
				Step := 10;
			ELSIF DirCreate_0.status <> ERR_FUB_BUSY THEN
				Status := DirCreate_0.status;
				Step := 0;
			END_IF
		9: // Try to delete the html file. This is necessary, because of when settings are changed, the file needs to be recreated.
			FileDelete_0(enable := TRUE, pDevice := ADR(FileDevUser), pName := ADR(FileNameVisImgHtml));
			IF FileDelete_0.status = ERR_OK OR FileDelete_0.status = fiERR_FILE_NOT_FOUND THEN
				Step := 10;
			ELSIF FileDelete_0.status <> ERR_FUB_BUSY THEN
				Status := FileDelete_0.status;
				Step := 0;
			END_IF
		10: // Check if html page exists
			FileCreate_0(enable := TRUE, pDevice := ADR(FileDevUser), pFile := ADR(FileNameVisImgHtml));
			IF FileCreate_0.status = ERR_OK THEN
				brsstrcpy(ADR(FileWriteData), ADR(HtmlFileContent1));
				brsstrcat(ADR(FileWriteData), ADR(EthIP));
				brsstrcat(ADR(FileWriteData), ADR(HtmlFileContent2));
				Step := 11;
			ELSIF FileCreate_0.status = fiERR_EXIST THEN
				Step := 20;
			ELSIF FileCreate_0.status <> ERR_FUB_BUSY THEN
				Status := FileCreate_0.status;
				Step := 0;
			END_IF
		11: // Write content
			FileWrite_0(enable := TRUE, ident := FileCreate_0.ident, offset := 0, pSrc := ADR(FileWriteData), len := brsstrlen(ADR(FileWriteData)));
			IF FileWrite_0.status = ERR_OK THEN
				Step := 12;
			ELSIF FileWrite_0.status <> ERR_FUB_BUSY THEN
				Status := FileWrite_0.status;
				Step := 0;
			END_IF
		12: // Close file
			FileClose_0(enable := TRUE, ident := FileCreate_0.ident);
			IF FileClose_0.status = ERR_OK THEN
				Step := 20;
			ELSIF FileClose_0.status <> ERR_FUB_BUSY THEN
				Status := FileClose_0.status;
				Step := 0;
			END_IF

		20: // Create FileDevice to System partition
			DevLink_0(enable := TRUE, pDevice := ADR(FileDevSystem), pParam := ADR(FileDevSystemPara));
			IF DevLink_0.status = ERR_OK THEN
				Step := 21;
			ELSIF DevLink_0.status <> ERR_FUB_BUSY THEN
				Status := DevLink_0.status;
				Step := 0;
			END_IF
		21: // Copy VisionEye.png from mappView folder (System partition) to webserver dir
			FileCopy_0(enable := TRUE, pSrcDev := ADR(FileDevSystem), pSrc := ADR(FileNameEyeSystem), pDestDev := ADR(FileDevUser), pDest := ADR(FileNameEyeUser));
			IF FileCopy_0.status <> ERR_FUB_BUSY THEN
				Status := FileCopy_0.status;
				Step := 22;
			END_IF
		22: // Delete DevLink
			DevUnlink_0(enable := TRUE, handle := DevLink_0.handle);
			IF DevUnlink_0.status = ERR_OK THEN
				Step := 30;
			ELSIF DevUnlink_0.status <> ERR_FUB_BUSY THEN
				Status := DevUnlink_0.status;
				Step := 0;
			END_IF
		30: // Create path for webviewer widget
			visWebViewerPath := 'http://'; // Create path for webviewer widget
			brsstrcat(ADR(visWebViewerPath), ADR(EthIP));
			Done := TRUE;
			Status := ERR_OK;
			Step := 0;
	END_CASE
END_FUNCTION_BLOCK
```

#### ViDownloadImage.st - not listed in the package file held
```iecst
// Note: This FBK needs to be called at least once in the INIT of the task to alloc memory (restriction of AsMem)
FUNCTION_BLOCK ViDownloadImage
	IF MemSvgAdr = 0 THEN // This will only be done once in the INIT of the task
		// Create memory for saving the image
		// Size: a 5MP picture in bmp format has less than 6.000.000 Bytes. A SVG with bas64 conversion maximum the 4/3 size.
		// UploadSize					:= 6000000;		// Upload of the picture data with httpClient
		// SvgHeaderSize				:= 2000; 		// Fileheader, ...
		// CrosshSize					:= 18000; 		// Crosshairs, Texts, ...
		MemSvgSize						:= 6000000 * 4 / 3 + 2000 + 18000;
		AsMemPartCreate_0.enable		:= TRUE;
		AsMemPartCreate_0.len			:= MemSvgSize + 1000; // 1000 Bytes for AsMemPart stuff/header
		AsMemPartCreate_0();
		IF AsMemPartCreate_0.status = ERR_OK THEN
			// Svg mem for creating the svg file including the image
			AsMemPartAllocClear_0.len	:= MemSvgSize;
			AsMemPartAllocClear_0(enable := TRUE, ident := AsMemPartCreate_0.ident);
			IF AsMemPartAllocClear_0.status = ERR_OK THEN
				MemSvgAdr 				:= AsMemPartAllocClear_0.mem;
			END_IF
		END_IF
	END_IF
	IF NOT Enable THEN
		Status := ERR_FUB_ENABLE_FALSE;
		Step := 0;
		RETURN;
	END_IF
	CASE Step OF
		0:
			visDownloadFileUrl := '';
			Status := ERR_FUB_BUSY;
			IF MemSvgAdr <> 0 THEN
				Step := 1;
			END_IF
		1:
			FileOpen_0.enable	:= TRUE;
			FileOpen_0.pDevice 	:= ADR(FileDevice);
			FileOpen_0.pFile	:= ADR(FileName);
			FileOpen_0();
			IF FileOpen_0.status = ERR_OK THEN
				IF FileOpen_0.filelen <= MemSvgSize THEN // Make sure file fits into memory
					brsmemset(MemSvgAdr, 0, MemSvgSize);
					Step := 2;
				ELSE // File is too large
					Status := ERR_MEM_DOWNLOAD;
					Step := 0;
				END_IF
			ELSIF FileOpen_0.status <> ERR_FUB_BUSY THEN
				Status := FileOpen_0.status;
				Step := 0;
			END_IF
		2:
			FileRead_0.enable	:= TRUE;
			FileRead_0.ident	:= FileOpen_0.ident;
			FileRead_0.len		:= FileOpen_0.filelen;
			FileRead_0.pDest	:= MemSvgAdr;
			FileRead_0();
			IF FileRead_0.status = ERR_OK THEN
				Step := 3;
			ELSIF FileRead_0.status <> ERR_FUB_BUSY THEN
				Status := FileRead_0.status;
				Step := 0;
			END_IF
		3:
			FileClose_0.enable	:= TRUE;
			FileClose_0.ident	:= FileOpen_0.ident;
			FileClose_0();
			IF FileClose_0.status = ERR_OK THEN
				Step := 4;
			ELSIF FileClose_0.status <> ERR_FUB_BUSY THEN
				Status := FileClose_0.status;
				Step := 0;
			END_IF
		4:
			TON_Timeout(IN := FALSE);
			httpService_Download(enable := FALSE, send := FALSE);
			IF httpService_Download.status = ERR_FUB_ENABLE_FALSE THEN
				Step := 5;
			END_IF
		5:
			// Create response header
			response_header_data :=  'Content-Type: application/octet-stream; Content-Transfer-Encoding: binary; Content-Disposition: attachment; filename="';
			brsstrcat(ADR(response_header_data), ADR(ImgName));
			brsstrcat(ADR(response_header_data), ADR('"'));
			// Pre-configure web service for download
			response_header.rawHeader.pData 	:= ADR(response_header_data);
			response_header.rawHeader.dataSize 	:= SIZEOF(response_header_data);
			response_header.rawHeader.dataLen 	:= brsstrlen(ADR(response_header_data));
			// Start web service
			httpService_Download.enable 			:= TRUE;
			httpService_Download.option 			:= httpOPTION_HTTP_10 + httpOPTION_SERVICE_TYPE_NAME;
			httpService_Download.pResponseData 		:= MemSvgAdr;
			httpService_Download.pResponseHeader	:= ADR(response_header);
			httpService_Download.pServiceName 		:= ADR(ImgName);
			httpService_Download.responseDataLen 	:= FileOpen_0.filelen;
			httpService_Download();

			// Timeout if file is not pulled from browser
			TON_Timeout(IN := TRUE, PT := T#3s);
			IF TON_Timeout.Q THEN
				Status := ERR_TIMEOUT_DOWNLOAD;
				Step := 0;
			END_IF

			IF httpService_Download.status = ERR_FUB_BUSY AND visDownloadFileUrl = '' THEN // Set URL
				brsstrcpy(ADR(visDownloadFileUrl), ADR(ImgName));
			ELSIF httpService_Download.status = ERR_OK AND NOT httpService_Download.send AND visDownloadFileUrl <> '' THEN // Start sending data
				httpService_Download.send := TRUE;
			ELSIF httpService_Download.send THEN // Sending data in progress
				Step := 6;
			ELSIF httpService_Download.status <> ERR_FUB_BUSY AND httpService_Download.status <> 0 THEN // Error
				Status := httpService_Download.status;
				Step := 0;
			END_IF

		6: // Wait until download is ready
			httpService_Download();
			TON_Timeout(IN := TRUE, PT := T#3s);
			IF TON_Timeout.Q THEN
				Status := ERR_TIMEOUT_DOWNLOAD;
				Step := 0;
			END_IF

			IF httpService_Download.phase = httpPHASE_WAITING THEN
				httpService_Download.send := FALSE;
				Status := 0;
				Step := 0;
			ELSIF httpService_Download.status <> ERR_FUB_BUSY THEN
				Status := httpService_Download.status;
				Step := 0;
			END_IF
		100:
	END_CASE
END_FUNCTION_BLOCK
```

#### ViDrawCrosshair.st - not listed in the package file held
```iecst
FUNCTION_BLOCK ViDrawCrosshair
	// Assign pointers
	IF VisionSensor.CFG.DataStructure <> 0 THEN
		CASE VisionSensor.CFG.VisionFunction OF
			enumBlob:
				Blob ACCESS VisionSensor.CFG.DataStructure;
			enumCoderReader:
				CodeReader ACCESS VisionSensor.CFG.DataStructure;
			enumMatch:
				Match ACCESS VisionSensor.CFG.DataStructure;
			enumMeasurement:
				MT ACCESS VisionSensor.CFG.DataStructure;
			enumOCR:
				OCR ACCESS VisionSensor.CFG.DataStructure;
			enumPixelCounter:
				Pixel ACCESS VisionSensor.CFG.DataStructure;
		END_CASE
	ELSE
		RETURN;
	END_IF

	// Draw cross hairs
	IF CmdRefreshCrosshair OR (visCrossHair.ShowCrosshair <> ShowCrosshairOld) OR (visCrossHair.DetailsNo <> DetailsNoOld) OR (SelectedSensor <> SelectedSensorOld) OR (ImageRotation_deg <> ImageRotation_degOld) OR (TextAlignment <> TextAlignmentOld) THEN
		ShowCrosshairOld		:= visCrossHair.ShowCrosshair;
		SelectedSensorOld		:= SelectedSensor;
		ImageRotation_degOld	:= ImageRotation_deg;
		TextAlignmentOld		:= TextAlignment;
		// First delete transformation and make everything invisible
		brsmemset(ADR(visCrossHair.SvgTransformation), 0, SIZEOF(visCrossHair.SvgTransformation));
		brsmemset(ADR(visCrossHair.SvgVisible), 0, SIZEOF(visCrossHair.SvgVisible));
		IF visCrossHair.ShowCrosshair THEN
			// Handle details no
			IF visCrossHair.DetailsNo < 1 THEN
				IF VisionSensor.DAT.ResultCnt > 0 THEN
					visCrossHair.DetailsNo := VisionSensor.DAT.ResultCnt;
				ELSE
					visCrossHair.DetailsNo := 1;
				END_IF
			END_IF
			IF visCrossHair.DetailsNo > VisionSensor.DAT.ResultCnt THEN
				visCrossHair.DetailsNo := 1;
			END_IF
			DetailsNoOld := visCrossHair.DetailsNo;

			// Create cross hairs and data for all results
			FOR idx := 1 TO MAX_NUM_RESULTS DO
				ResultModelNumber	:= 0;
				ResultPositionX		:= 0;
				ResultPositionY		:= 0;
				ResultOrientation	:= 0;
				brsmemset(ADR(CrossHairInfo[idx]), 0, SIZEOF(CrossHairInfo[0]));

				// Make sure we have data to display
				IF VisionSensor.DAT.ResultCnt <> 0 AND idx <= VisionSensor.DAT.ResultCnt THEN
					// Select data source from vision function
					MT_UseXY := FALSE;
					CASE VisionSensor.CFG.VisionFunction OF
						enumBlob:
							ResultModelNumber	:= Blob.ModelNumber[idx];
							ResultPositionX		:= UDINT_TO_REAL(Blob.PositionX[idx]) / visCrossHair.CFG.PixelRatio;
							ResultPositionY		:= UDINT_TO_REAL(Blob.PositionY[idx]) / visCrossHair.CFG.PixelRatio;
							ResultOrientation	:= Blob.Orientation[idx] / visCrossHair.CFG.PixelRatio;
						enumPixelCounter:
							ResultModelNumber	:= Pixel.ModelNumber[idx];
							ResultPositionX		:= UDINT_TO_REAL(Pixel.PositionX[idx]) / visCrossHair.CFG.PixelRatio;
							ResultPositionY		:= UDINT_TO_REAL(Pixel.PositionY[idx]) / visCrossHair.CFG.PixelRatio;
						enumCoderReader:
							ResultPositionX		:= UDINT_TO_REAL(CodeReader.PositionX[idx]) / visCrossHair.CFG.PixelRatio;
							ResultPositionY		:= UDINT_TO_REAL(CodeReader.PositionY[idx]) / visCrossHair.CFG.PixelRatio;
							ResultOrientation	:= CodeReader.Orientation[idx] / visCrossHair.CFG.PixelRatio;
						enumMatch:
							ResultModelNumber	:= Match.ModelNumber[idx];
							ResultPositionX		:= UDINT_TO_REAL(Match.PositionX[idx]) / visCrossHair.CFG.PixelRatio;
							ResultPositionY		:= UDINT_TO_REAL(Match.PositionY[idx]) / visCrossHair.CFG.PixelRatio;
							ResultOrientation	:= Match.Orientation[idx] / visCrossHair.CFG.PixelRatio;
						enumMeasurement:
							IF MT.UseResultAsXY THEN
								ResultPositionX	:= UDINT_TO_REAL(MT.Result[idx])/10;
								ResultPositionY	:= UDINT_TO_REAL(MT.Result[idx+1])/10;
								idx := idx + 1;
							END_IF
							MT_UseXY := TRUE; // use this variable because of in case Visionfunction != MT then the Pointer MT is not initialized
						enumOCR:
							ResultPositionX		:= UDINT_TO_REAL(OCR.PositionX[idx]) / visCrossHair.CFG.PixelRatio;
							ResultPositionY		:= UDINT_TO_REAL(OCR.PositionY[idx]) / visCrossHair.CFG.PixelRatio;
							ResultOrientation	:= OCR.Orientation[idx] / visCrossHair.CFG.PixelRatio;
					END_CASE

					// Adapt the size to the size of the WebViewer image in mapp View. The download as svg file also uses a fixed size (both 1280x1024)
					ResultPositionX				:= ResultPositionX * UINT_TO_REAL(visCrossHair.CFG.RefSizeX) / UINT_TO_REAL(VisionSensor.CFG.ResolutionWidth_X);
					ResultPositionY				:= ResultPositionY * UINT_TO_REAL(visCrossHair.CFG.RefSizeY) / UINT_TO_REAL(VisionSensor.CFG.ResolutionHeight_Y);

					// Show crosshair except for measurement function
					IF VisionSensor.CFG.VisionFunction <> enumMeasurement OR MT_UseXY THEN
						IF ResultPositionX <> 0 AND ResultPositionY <> 0 THEN
							visCrossHair.SvgVisible[idx] := TRUE;

							// Calculate cross information, also needed for saving the svg in ViSaveImgOnPLC
							CrossHairInfo[idx].CrosshairScale			:= visCrossHair.CFG.Scale;
							CrossHairInfo[idx].CrosshairSizeScaled		:= USINT_TO_REAL(visCrossHair.CFG.Size) * visCrossHair.CFG.Scale;
							CrossHairInfo[idx].CrosshairTopLeftX		:= ResultPositionX - CrossHairInfo[idx].CrosshairSizeScaled / 2.0;
							CrossHairInfo[idx].CrosshairTopLeftY		:= ResultPositionY - CrossHairInfo[idx].CrosshairSizeScaled / 2.0;
							CrossHairInfo[idx].CrosshairRotateCenter	:= ResultOrientation * -1;

							// Crosshair transformation for displaying in the mappView visu
							IF visCrossHair.DetailsNo = idx THEN
								svgTrafo := '[{"select":"#CrosshairBlue","display":false}, {"select":"#CrosshairRed","display":true, "translate":[';
							ELSE
								svgTrafo := '[{"select":"#CrosshairRed","display":false}, { "select":"#CrosshairBlue","display":true, "translate":[';
							END_IF
							// Crosshair position
							CrosshSize		:= CrossHairInfo[idx].CrosshairSizeScaled / 2.0;
							ScaleVertical	:= UINT_TO_REAL(VisionSensor.CFG.ResolutionHeight_Y) / UINT_TO_REAL(VisionSensor.CFG.ResolutionWidth_X);
							CASE ImageRotation_deg OF
								0:		brsitoa(REAL_TO_INT(ResultPositionX															- CrosshSize), ADR(tmpStr));
								90:		brsitoa(REAL_TO_INT((VisionSensor.CFG.ResolutionHeight_Y - ResultPositionY) * ScaleVertical	- CrosshSize), ADR(tmpStr));
								180:	brsitoa(REAL_TO_INT(VisionSensor.CFG.ResolutionWidth_X - ResultPositionX					- CrosshSize), ADR(tmpStr));
								270:	brsitoa(REAL_TO_INT(ResultPositionY * ScaleVertical											- CrosshSize), ADR(tmpStr));
							ELSE
										brsitoa(REAL_TO_INT(ResultPositionX															- CrosshSize), ADR(tmpStr));
							END_CASE
							brsstrcat(ADR(svgTrafo), ADR(tmpStr));
							brsstrcat(ADR(svgTrafo), ADR(','));
							CASE ImageRotation_deg OF
								0:		brsitoa(REAL_TO_INT(ResultPositionY															- CrosshSize), ADR(tmpStr));
								90:		brsitoa(REAL_TO_INT(ResultPositionX * ScaleVertical											- CrosshSize), ADR(tmpStr));
								180:	brsitoa(REAL_TO_INT(VisionSensor.CFG.ResolutionHeight_Y - ResultPositionY					- CrosshSize), ADR(tmpStr));
								270:	brsitoa(REAL_TO_INT((VisionSensor.CFG.ResolutionWidth_X - ResultPositionX) * ScaleVertical	- CrosshSize), ADR(tmpStr));
							ELSE
										brsitoa(REAL_TO_INT(ResultPositionY															- CrosshSize), ADR(tmpStr));
							END_CASE
							brsstrcat(ADR(svgTrafo), ADR(tmpStr));
							// Add cross hair scaling
							brsstrcat(ADR(svgTrafo), ADR('],"scale":['));
							brsftoa(visCrossHair.CFG.Scale, ADR(tmpStr));
							brsstrcat(ADR(svgTrafo), ADR(tmpStr));
							brsstrcat(ADR(svgTrafo), ADR(','));
							brsstrcat(ADR(svgTrafo), ADR(tmpStr));
							// Add cross hair rotation
							brsstrcat(ADR(svgTrafo), ADR('],"spin":['));
							brsftoa(CrossHairInfo[idx].CrosshairRotateCenter - ImageRotation_deg, ADR(tmpStr));
							brsstrcat(ADR(svgTrafo), ADR(tmpStr));
							brsstrcat(ADR(svgTrafo), ADR(','));
							brsftoa(USINT_TO_REAL(visCrossHair.CFG.Size) / 2, ADR(tmpStr)); // For mappView the rotation is based on the original size, not on the scaled size
							brsstrcat(ADR(svgTrafo), ADR(tmpStr));
							brsstrcat(ADR(svgTrafo), ADR(','));
							brsstrcat(ADR(svgTrafo), ADR(tmpStr));
							brsstrcat(ADR(svgTrafo), ADR(']}]'));
							visCrossHair.SvgTransformation[idx] := svgTrafo;

							// Add text data to selected cross hair (small index number)
							IF visCrossHair.DetailsNo = idx THEN
								svgContent := '<text class="cText" fill="red " font-size="22" font-family="Helvetica, Arial, sans-serif"><tspan class="text" x="';
							ELSE
								svgContent := '<text class="cText" fill="blue" font-size="22" font-family="Helvetica, Arial, sans-serif"><tspan class="text" x="';
							END_IF
							CASE ImageRotation_deg OF
								0:		brsitoa(REAL_TO_INT(ResultPositionX															+ CrosshSize), ADR(tmpStr));
								90:		brsitoa(REAL_TO_INT((VisionSensor.CFG.ResolutionHeight_Y - ResultPositionY) * ScaleVertical	+ CrosshSize), ADR(tmpStr));
								180:	brsitoa(REAL_TO_INT(VisionSensor.CFG.ResolutionWidth_X - ResultPositionX					+ CrosshSize), ADR(tmpStr));
								270:	brsitoa(REAL_TO_INT(ResultPositionY * ScaleVertical											+ CrosshSize), ADR(tmpStr));
							ELSE
										brsitoa(REAL_TO_INT(ResultPositionX															+ CrosshSize), ADR(tmpStr));
							END_CASE
							brsstrcat(ADR(svgContent), ADR(tmpStr));
							brsstrcat(ADR(svgContent), ADR('" y="'));
							CASE ImageRotation_deg OF
								0:		brsitoa(REAL_TO_INT(ResultPositionY															+ 5), ADR(tmpStr));
								90:		brsitoa(REAL_TO_INT(ResultPositionX * ScaleVertical											+ 5), ADR(tmpStr));
								180:	brsitoa(REAL_TO_INT(VisionSensor.CFG.ResolutionHeight_Y - ResultPositionY					+ 5), ADR(tmpStr));
								270:	brsitoa(REAL_TO_INT((VisionSensor.CFG.ResolutionWidth_X - ResultPositionX) * ScaleVertical	+ 5), ADR(tmpStr));
							ELSE
										brsitoa(REAL_TO_INT(ResultPositionY															+ 5), ADR(tmpStr));
							END_CASE
							brsstrcat(ADR(svgContent), ADR(tmpStr));
							brsstrcat(ADR(svgContent), ADR('"> '));
							// Add result number
							brsitoa(idx, ADR(tmpStr));
							brsstrcat(ADR(svgContent), ADR(tmpStr));
							brsstrcat(ADR(svgContent), ADR('</tspan></text>'));

							// for saving svg file. The texts added below are not of interest for the saved SVG, so copy it now before adding the details information
							brsstrcpy(ADR(CrossHairInfo[idx].Text), ADR(svgContent));
							blueTextPos := FIND(CrossHairInfo[idx].Text, 'fill="blue"'); // Make all texts red. In the SVG is no highlighted crosshair
							IF blueTextPos > 2 THEN
								brsmemcpy(ADR(CrossHairInfo[idx].Text) + blueTextPos - 1, ADR('fill="red "'), 11);
							END_IF
							visCrossHair.SvgContent[idx] := svgContent;

							// Create details information to show in the top left or right corner
							brsstrcat(ADR(svgContent), ADR('<text class="cText" fill="red" font-size="35" font-family="Helvetica, Arial, sans-serif" x="10" y="10"> '));
							CrossHairInfo[1].DataVis	:= '';
							CrossHairInfo[idx].Data		:= '';
							// Add model ID information for blob and match
							IF VisionSensor.CFG.VisionFunction = enumBlob OR VisionSensor.CFG.VisionFunction = enumMatch THEN
								CrosshairDetailsValue(ADR(svgContent),  ADR('Model ID: '), ResultModelNumber, TextAlignment);
								brsstrcat(ADR(CrossHairInfo[1].DataVis), ADR('1, '));
								brsitoa(ResultModelNumber, ADR(tmpStr));
								brsstrcat(ADR(CrossHairInfo[idx].Data), ADR(tmpStr));
								brsstrcat(ADR(CrossHairInfo[idx].Data), ADR(', '));
							ELSE
								brsstrcat(ADR(CrossHairInfo[1].DataVis), ADR('0, '));
								brsstrcat(ADR(CrossHairInfo[idx].Data), ADR('"none", '));
							END_IF
							// Add X and Y position information
							CrosshairDetailsValue(ADR(svgContent),  ADR('Pos X: '), ResultPositionX, TextAlignment);
							CrosshairDetailsValue(ADR(svgContent),  ADR('Pos Y: '), ResultPositionY, TextAlignment);
							brsstrcat(ADR(CrossHairInfo[1].DataVis), ADR('1, 1, '));
							brsftoa(ResultPositionX, ADR(tmpStr));
							brsstrcat(ADR(CrossHairInfo[idx].Data), ADR(tmpStr));
							brsstrcat(ADR(CrossHairInfo[idx].Data), ADR(', '));
							brsftoa(ResultPositionY, ADR(tmpStr));
							brsstrcat(ADR(CrossHairInfo[idx].Data), ADR(tmpStr));
							brsstrcat(ADR(CrossHairInfo[idx].Data), ADR(', '));
							// Add orientation information
							IF VisionSensor.CFG.VisionFunction <> enumMeasurement THEN
								CrosshairDetailsValue(ADR(svgContent),  ADR('Orientation: '), ResultOrientation, TextAlignment);
								brsstrcat(ADR(CrossHairInfo[1].DataVis), ADR('1, '));
								brsftoa(ResultOrientation, ADR(tmpStr));
								brsstrcat(ADR(CrossHairInfo[idx].Data), ADR(tmpStr));
								brsstrcat(ADR(CrossHairInfo[idx].Data), ADR(', '));
							ELSE
								brsstrcat(ADR(CrossHairInfo[1].DataVis), ADR('0, '));
								brsstrcat(ADR(CrossHairInfo[idx].Data), ADR('"none", '));
							END_IF
							// Add detail information for blob
							IF VisionSensor.CFG.VisionFunction = enumBlob THEN
								IF Blob.EnhancedBlobInformation = 1 THEN // Only access the Pointer Blob if it really exists. So don't combine this line of code with the line before
									CrosshairDetailsValue(ADR(svgContent),  ADR('Clipped: '), Blob.Clipped[idx], TextAlignment);
									CrosshairDetailsValue(ADR(svgContent),  ADR('Gray: '), Blob.MeanGrayValue[idx], TextAlignment);
									CrosshairDetailsValue(ADR(svgContent),  ADR('Length: '), UDINT_TO_REAL(Blob.Length[idx])/visCrossHair.CFG.PixelRatio, TextAlignment);
									CrosshairDetailsValue(ADR(svgContent),  ADR('Width: '), UDINT_TO_REAL(Blob.Width[idx])/visCrossHair.CFG.PixelRatio, TextAlignment);
									CrosshairDetailsValue(ADR(svgContent),  ADR('Area: '), UDINT_TO_REAL(Blob.Area[idx])/visCrossHair.CFG.PixelRatio, TextAlignment);
									brsstrcat(ADR(CrossHairInfo[1].DataVis), ADR('1, 1, 1, 1, 1, '));
									brsitoa(Blob.Clipped[idx], ADR(tmpStr));
									brsstrcat(ADR(CrossHairInfo[idx].Data), ADR(tmpStr));
									brsstrcat(ADR(CrossHairInfo[idx].Data), ADR(', '));
									brsitoa(Blob.MeanGrayValue[idx], ADR(tmpStr));
									brsstrcat(ADR(CrossHairInfo[idx].Data), ADR(tmpStr));
									brsstrcat(ADR(CrossHairInfo[idx].Data), ADR(', '));
									brsftoa(UDINT_TO_REAL(Blob.Length[idx])/visCrossHair.CFG.PixelRatio, ADR(tmpStr));
									brsstrcat(ADR(CrossHairInfo[idx].Data), ADR(tmpStr));
									brsstrcat(ADR(CrossHairInfo[idx].Data), ADR(', '));
									brsftoa(UDINT_TO_REAL(Blob.Width[idx])/visCrossHair.CFG.PixelRatio, ADR(tmpStr));
									brsstrcat(ADR(CrossHairInfo[idx].Data), ADR(tmpStr));
									brsstrcat(ADR(CrossHairInfo[idx].Data), ADR(', '));
									brsftoa(UDINT_TO_REAL(Blob.Area[idx])/visCrossHair.CFG.PixelRatio, ADR(tmpStr));
									brsstrcat(ADR(CrossHairInfo[idx].Data), ADR(tmpStr));
									brsstrcat(ADR(CrossHairInfo[idx].Data), ADR(', '));
								ELSE
									brsstrcat(ADR(CrossHairInfo[1].DataVis), ADR('0, 0, 0, 0, 0, '));
									brsstrcat(ADR(CrossHairInfo[idx].Data), ADR('"none", "none", "none", "none", "none", '));
								END_IF
							ELSE
								brsstrcat(ADR(CrossHairInfo[1].DataVis), ADR('0, 0, 0, 0, 0, '));
								brsstrcat(ADR(CrossHairInfo[idx].Data), ADR('"none", "none", "none", "none", "none", '));
							END_IF
							// Add detail information for match
							IF VisionSensor.CFG.VisionFunction = enumMatch THEN
								CrosshairDetailsValue(ADR(svgContent),  ADR('Score: '), Match.Score[idx], TextAlignment);
								CrosshairDetailsValue(ADR(svgContent),  ADR('Scale: '), Match.Scale[idx], TextAlignment);
								brsstrcat(ADR(CrossHairInfo[1].DataVis), ADR('1, 1, '));
								brsitoa(Match.Score[idx], ADR(tmpStr));
								brsstrcat(ADR(CrossHairInfo[idx].Data), ADR(tmpStr));
								brsstrcat(ADR(CrossHairInfo[idx].Data), ADR(', '));
								brsitoa(Match.Scale[idx], ADR(tmpStr));
								brsstrcat(ADR(CrossHairInfo[idx].Data), ADR(tmpStr));
								brsstrcat(ADR(CrossHairInfo[idx].Data), ADR(', '));
							ELSE
								brsstrcat(ADR(CrossHairInfo[1].DataVis), ADR('0, 0, '));
								brsstrcat(ADR(CrossHairInfo[idx].Data), ADR('"none", "none", '));
							END_IF
							// Add detail information for OCR and CodeReader
							IF VisionSensor.CFG.VisionFunction = enumOCR THEN
								CrosshairDetailsValue(ADR(svgContent),  ADR('Grading: '), OCR.Grading[idx], TextAlignment);
								CrosshairDetailsText(ADR(svgContent),  ADR('Text: '), ADR(OCR.Text[idx]), TextAlignment);
								brsstrcat(ADR(CrossHairInfo[1].DataVis), ADR('1, 0, 1, ')); // Grading, Code Type, Text
								brsitoa(OCR.Grading[idx], ADR(tmpStr));
								brsstrcat(ADR(CrossHairInfo[idx].Data), ADR(tmpStr));
								brsstrcat(ADR(CrossHairInfo[idx].Data), ADR(', "none", "'));
								brsstrcat(ADR(CrossHairInfo[idx].Data), ADR(OCR.Text[idx]));
								brsstrcat(ADR(CrossHairInfo[idx].Data), ADR('", '));
							ELSIF VisionSensor.CFG.VisionFunction = enumCoderReader THEN
								CrosshairDetailsText(ADR(svgContent),  ADR('Code: '), ADR(CodeTypes[LIMIT(0, CodeReader.BarcodeType[idx], MAX_NUM_CODETYPES)]), TextAlignment);
								CrosshairDetailsText(ADR(svgContent),  ADR('Text: '), ADR(CodeReader.BarcodeText[idx]), TextAlignment);
								brsstrcat(ADR(CrossHairInfo[1].DataVis), ADR('0, 1, 1, ')); // Grading, Code Type, Text
								brsstrcat(ADR(CrossHairInfo[idx].Data), ADR('"none", "'));
								brsstrcat(ADR(CrossHairInfo[idx].Data), ADR(CodeTypes[LIMIT(0, CodeReader.BarcodeType[idx], MAX_NUM_CODETYPES)]));
								brsstrcat(ADR(CrossHairInfo[idx].Data), ADR('", "'));
								brsstrcat(ADR(CrossHairInfo[idx].Data), ADR(CodeReader.BarcodeText[idx]));
								brsstrcat(ADR(CrossHairInfo[idx].Data), ADR('", '));
							ELSE
								brsstrcat(ADR(CrossHairInfo[1].DataVis), ADR('0, 0, 0, '));
								brsstrcat(ADR(CrossHairInfo[idx].Data), ADR('"none", "none", "none", '));
							END_IF
							brsstrcat(ADR(CrossHairInfo[1].DataVis), ADR('0')); // For the not used "Result"
							brsstrcat(ADR(CrossHairInfo[idx].Data), ADR('"none"')); // For the not used "Result"
							brsstrcat(ADR(svgContent), ADR('</text>'));
							// Add text data from selected cross hair in the top left corner of the image, but only if the index is the actual index
							IF visCrossHair.DetailsNo = idx THEN
								visCrossHair.SvgContent[idx] := svgContent;
							END_IF
						END_IF
					ELSE // Add result information for measurement
						visCrossHair.SvgTransformation[idx] := '[{"select":"#CrosshairRed","display":false}, {"select":"#CrosshairBlue","display":false}]';
						visCrossHair.SvgVisible[idx] := TRUE;
						brsstrcpy(ADR(svgContent), ADR('<text class="cText" fill="red" font-size="35" font-family="Helvetica, Arial, sans-serif" x="10" y="'));
						brsitoa(idx*40, ADR(tmpStr));
						brsstrcat(ADR(svgContent), ADR(tmpStr));
						brsstrcat(ADR(svgContent), ADR('"> '));
						CrosshairDetailsValue(ADR(svgContent),  ADR('Result:'), UDINT_TO_REAL(MT.Result[idx])/1000, TextAlignment);
						brsstrcat(ADR(svgContent), ADR('</text>'));
						visCrossHair.SvgContent[idx] := svgContent;
						brsstrcpy(ADR(CrossHairInfo[1].DataVis), ADR('0, 0, 0, 0, 0, 0, 0, 0, 0, 0, 0, 0, 0, 0, 1'));
						brsstrcpy(ADR(CrossHairInfo[idx].Data), ADR('"none", "none", "none", "none", "none", "none", "none", "none", "none", "none", "none", "none", "none", "none", '));
						brsftoa(UDINT_TO_REAL(MT.Result[idx])/1000, ADR(tmpStr));
						brsstrcat(ADR(CrossHairInfo[idx].Data), ADR(tmpStr));
					END_IF
				ELSIF VisionSensor.DAT.ResultCnt = 0 AND VisionDisabled THEN // Vision function is disabled --> show a message
					visCrossHair.SvgVisible[1]			:= TRUE;
					visCrossHair.SvgTransformation[1]	:= '[{"select":"#CrosshairRed","display":false}, {"select":"#CrosshairBlue","display":false}]';
					visCrossHair.SvgContent[1]			:= '<text class="cText" fill="red" font-size="35" font-family="Helvetica, Arial, sans-serif" x="10" y="40"> Processing is disabled </text>';
				END_IF
			END_FOR
		END_IF // IF visCrossHair.ShowCrosshair THEN
	END_IF
END_FUNCTION_BLOCK
```

#### ViRefreshImageList.st - not listed in the package file held
```iecst
FUNCTION_BLOCK ViRefreshImageList
	IF NOT Enable THEN
		Status := ERR_FUB_ENABLE_FALSE;
		Step := 0;
		RETURN;
	END_IF
	CASE Step OF
		0:
			Status := ERR_FUB_BUSY;
			Step := 1;
		1: // Reset everything
			brsmemset(ADR(VisionImage.DAT.Images), 0, SIZEOF(VisionImage.DAT.Images));
			brsmemset(ADR(ImageList), 0, SIZEOF(ImageList));
			brsmemset(ADR(visSelectedImage), 0, SIZEOF(visSelectedImage));
			visSelectedImageOld := '';
			visSelectedImage	:= '';
			DirEntries			:= 0;
			idx					:= 0;
			file_newest			:= '';
			file_oldest			:= '';
			date_newest			:= UDINT_TO_DT(0);
			date_oldest			:= DT#2100-06-06-12:00:00;
			cmdDeleteOldest		:= FALSE;
			Step := 2;
		2: // Proceed with next entry
			DirRead_0.enable 	:= TRUE;
			DirRead_0.pDevice 	:= ADR(VisionImage.CFG.FileDevice);
			DirRead_0.pPath		:= ADR(VisionImage.CFG.DirName);
			DirRead_0.entry 	:= idx;
			DirRead_0.option 	:= fiFILE;
			DirRead_0.pData 	:= ADR(dir_data);
			DirRead_0.data_len 	:= SIZEOF(dir_data);
			DirRead_0();
			IF DirRead_0.status = ERR_OK THEN
				// Make sure file is an image and we have space to store it
				IF  brsstrcmp(ADR(dir_data.Filename) + brsstrlen(ADR(dir_data.Filename)) - 4, ADR('.bmp')) = 0 OR
				    brsstrcmp(ADR(dir_data.Filename) + brsstrlen(ADR(dir_data.Filename)) - 4, ADR('.jpg')) = 0 OR
					brsstrcmp(ADR(dir_data.Filename) + brsstrlen(ADR(dir_data.Filename)) - 4, ADR('.svg')) = 0 THEN
					// Find newest and oldest file
					IF dir_data.Date > date_newest THEN
						brsstrcpy(ADR(file_newest), ADR(dir_data.Filename));
						date_newest := dir_data.Date;
					END_IF
					IF dir_data.Date < date_oldest THEN
						brsstrcpy(ADR(file_oldest), ADR(dir_data.Filename));
						date_oldest := dir_data.Date;
					END_IF
					IF DirEntries <= SIZEOF(ImageList)/SIZEOF(ImageList[0]) - 1 THEN
						brsstrcpy(ADR(VisionImage.DAT.Images[DirEntries]), ADR(dir_data.Filename));
						// Create list box data
						ImageList[DirEntries] := '{"value":"';
						brsstrcat(ADR(ImageList[DirEntries]), ADR(dir_data.Filename));
						brsstrcat(ADR(ImageList[DirEntries]), ADR('","text":"'));
						brsstrcat(ADR(ImageList[DirEntries]), ADR(dir_data.Filename));
						brsstrcat(ADR(ImageList[DirEntries]), ADR('"}'));
						DirEntries := DirEntries + 1;
					ELSE
						cmdDeleteOldest := TRUE; // the oldest needs to be deleted. But first we have to search for all images to detect the oldest image. So now don't change the step
					END_IF
				END_IF
				idx := idx + 1;
			ELSIF DirRead_0.status = fiERR_NO_MORE_ENTRIES THEN // Finish up when last entry was reached
				IF cmdDeleteOldest THEN // Delete oldest file if there are too many entries
					cmdDeleteOldest := FALSE;
					brsstrcpy(ADR(DeleteFileName), ADR(VisionImage.CFG.DirName));
					brsstrcat(ADR(DeleteFileName), ADR('/'));
					brsstrcat(ADR(DeleteFileName), ADR(file_oldest));
					Step := 10;
				ELSE
					TON_VisPause(IN := FALSE);
					Step := 3;
				END_IF
			ELSIF DirRead_0.status <> ERR_FUB_BUSY THEN
				Status := DirRead_0.status;
				Step := 0;
			END_IF
		3: // Wait for vis before setting last file
			TON_VisPause(IN := TRUE, PT := T#250ms);
			IF TON_VisPause.Q THEN
				brsstrcpy(ADR(visSelectedImage), ADR(file_newest));
				Status := 0;
				Step := 0;
			END_IF

		10: // Delete oldest image
			FileDelete_0.enable 	:= TRUE;
			FileDelete_0.pDevice	:= ADR(VisionImage.CFG.FileDevice);
			FileDelete_0.pName 		:= ADR(DeleteFileName);
			FileDelete_0();
			IF FileDelete_0.status = ERR_OK THEN
				Step := 0; // Refresh --> Read dir again, don't change the Status to 0!
			ELSIF FileDelete_0.status <> ERR_FUB_BUSY THEN
				Status := FileDelete_0.status;
				Step := 0;
			END_IF
	END_CASE
END_FUNCTION_BLOCK
```

#### ViSaveImgOnPlc.st - not listed in the package file held
```iecst
// Note: This FBK needs to be called at least once in the INIT of the task to alloc memory (restriction of AsMem)
FUNCTION_BLOCK ViSaveImgOnPlc
	IF MemInfo.SvgAdr = 0 THEN // This will only be done once in the INIT of the task
		// Create memory for uploading and transforming image
		// Size: a 5MP picture in bmp format has less than 6.000.000 Bytes. A SVG with bas64 conversion maximum the 4/3 size.
		MemInfo.UploadSize			:= 6000000;		// Upload of the picture data with httpClient
		MemInfo.SvgHeaderSize		:= 2000; 		// Fileheader, ...
		MemInfo.CrosshSize			:= 18000; 		// Crosshairs, Texts, ...
		MemInfo.SvgSize				:= MemInfo.UploadSize * 4 / 3 + MemInfo.SvgHeaderSize + MemInfo.CrosshSize;
		AsMemPartCreate_0.enable	:= TRUE;
		AsMemPartCreate_0.len		:= MemInfo.UploadSize + MemInfo.SvgSize + MemInfo.CrosshSize + 1000; // 1000 Bytes for AsMemPart stuff/header
		AsMemPartCreate_0();
		IF AsMemPartCreate_0.status = ERR_OK THEN
			// Upload mem for loading the image from camera to plc
			AsMemPartAllocClear_0.len		:= MemInfo.UploadSize;
			AsMemPartAllocClear_0(enable := TRUE, ident := AsMemPartCreate_0.ident);
			IF AsMemPartAllocClear_0.status = ERR_OK THEN
				MemInfo.UploadAdr			:= AsMemPartAllocClear_0.mem;
			END_IF
			// Svg mem for creating the svg file including the image
			AsMemPartAllocClear_0.len		:= MemInfo.SvgSize;
			AsMemPartAllocClear_0(enable := TRUE, ident := AsMemPartCreate_0.ident);
			IF AsMemPartAllocClear_0.status = ERR_OK THEN
				MemInfo.SvgAdr 				:= AsMemPartAllocClear_0.mem;
			END_IF
			// Mem for creating the crosshaurs
			AsMemPartAllocClear_0.len		:= MemInfo.CrosshSize;
			AsMemPartAllocClear_0(enable := TRUE, ident := AsMemPartCreate_0.ident);
			IF AsMemPartAllocClear_0.status = ERR_OK THEN
				MemInfo.CrosshAdr			:= AsMemPartAllocClear_0.mem;
			END_IF
		END_IF
	END_IF
	IF NOT Enable THEN
		Status := ERR_FUB_ENABLE_FALSE;
		Step := 0;
		RETURN;
	END_IF
	CASE Step OF
		0:
			Status := ERR_FUB_BUSY;
			IF MemInfo.UploadAdr <> 0 AND MemInfo.SvgAdr <> 0 AND MemInfo.CrosshAdr <> 0 THEN
				Step := 1;
			END_IF
		1: // Initialization
			ACTION_InitTexts;
			brsmemcpy(ADR(b64key), ADR('ABCDEFGHIJKLMNOPQRSTUVWXYZabcdefghijklmnopqrstuvwxyz0123456789+/'), SIZEOF(b64key));
			// Generate new filenames
			DTGetTime_0(enable := TRUE);
			DT_TO_DTStructure(DTGetTime_0.DT1, ADR(DTStructure_0));
			FileNameImg := CFG.DirName;
			brsstrcat(ADR(FileNameImg), ADR('/'));
			tmpStr1 := UINT_TO_STRING(DTStructure_0.year);
			brsstrcat(ADR(FileNameImg), ADR(tmpStr1));
			brsstrcat(ADR(FileNameImg), ADR('_'));
			tmpStr1 := USINT_TO_STRING(DTStructure_0.month);
			IF(DTStructure_0.month < 10) THEN
				brsstrcat(ADR(FileNameImg), ADR('0'));
			END_IF
			brsstrcat(ADR(FileNameImg), ADR(tmpStr1));
			brsstrcat(ADR(FileNameImg), ADR('_'));
			tmpStr1 := USINT_TO_STRING(DTStructure_0.day);
			IF(DTStructure_0.day < 10) THEN
				brsstrcat(ADR(FileNameImg), ADR('0'));
			END_IF
			brsstrcat(ADR(FileNameImg), ADR(tmpStr1));
			brsstrcat(ADR(FileNameImg), ADR('_'));
			tmpStr1 := USINT_TO_STRING(DTStructure_0.hour);
			IF(DTStructure_0.hour < 10) THEN
				brsstrcat(ADR(FileNameImg), ADR('0'));
			END_IF
			brsstrcat(ADR(FileNameImg), ADR(tmpStr1));
			brsstrcat(ADR(FileNameImg), ADR('_'));
			tmpStr1 := USINT_TO_STRING(DTStructure_0.minute);
			IF(DTStructure_0.minute < 10) THEN
				brsstrcat(ADR(FileNameImg), ADR('0'));
			END_IF
			brsstrcat(ADR(FileNameImg), ADR(tmpStr1));
			brsstrcat(ADR(FileNameImg), ADR('_'));
			tmpStr1 := USINT_TO_STRING(DTStructure_0.second);
			IF(DTStructure_0.second < 10) THEN
				brsstrcat(ADR(FileNameImg), ADR('0'));
			END_IF
			brsstrcat(ADR(FileNameImg), ADR(tmpStr1));
			brsstrcat(ADR(FileNameImg), ADR('.'));
			brsstrcpy(ADR(FileNameSvg), ADR(FileNameImg)); // Same filename but differend ending
			IF CFG.Format = 0 THEN
				brsstrcat(ADR(FileNameImg), ADR('jpg'));
			ELSE
				brsstrcat(ADR(FileNameImg), ADR('bmp'));
			END_IF
			brsstrcat(ADR(FileNameSvg), ADR('svg'));
			// Create URI and Host
			URI := '/';
			IF CFG.Format = 0 THEN
				brsstrcat(ADR(URI), ADR('jpg'));
				brsstrcat(ADR(URI), ADR('?q='));
				brsitoa(CFG.QualityJPG, ADR(tmpStr1));
				brsstrcat(ADR(URI), ADR(tmpStr1));
			ELSE
				brsstrcat(ADR(URI), ADR('bmp'));
			END_IF
			Host := CFG.PlkIPWithoutNode;
			brsitoa(PowerlinkNode, ADR(tmpStr1));
			brsstrcat(ADR(Host), ADR(tmpStr1));
			DiagStartTime := clock_ms();
			Step := 10;

		10: // Reset timer and HTTP client
			TON_ReloadTimeout(IN := FALSE);
			httpClient_0(enable := FALSE, abort := FALSE, send := FALSE);
			IF httpClient_0.status = ERR_FUB_ENABLE_FALSE THEN
				Step := 11;
			END_IF

		11: // Wait for response
			TON_ReloadTimeout(IN := TRUE, PT := T#10s); // Time out when no response after 10s
			RequestHeader.keepAlive			:= 'timeout=5, max=100';
			httpClient_0.enable				:= TRUE;
			httpClient_0.send				:= TRUE;
			httpClient_0.method 			:= httpMETHOD_GET;
			httpClient_0.option 			:= httpOPTION_HTTP_11;
			httpClient_0.hostPort			:= 8080;
			httpClient_0.pHost 				:= ADR(Host);
			httpClient_0.pUri 				:= ADR(URI);
			httpClient_0.pResponseData 		:= MemInfo.UploadAdr;
			httpClient_0.responseDataSize	:= MemInfo.UploadSize;
			httpClient_0.pRequestHeader		:= ADR(RequestHeader);
			httpClient_0();
			IF httpClient_0.status = ERR_OK AND httpClient_0.responseDataLen <> 0 THEN
				UploadedImgSize				:= httpClient_0.responseDataLen;
				httpClient_0(send := FALSE);
				IF UploadedImgSize < 100 THEN // No image available. Hint: In case of no image there will be sent 86 Bytes with an html error text
					Status := ERR_NO_IMAGE;
					Step := 0;
				ELSE
					IF CFG.UploadBmpJpg THEN
						Step := 20; // save the image (bmp or jpg)
					ELSE
						Step := 30; // directly upload the svg
					END_IF
				END_IF
			ELSIF httpClient_0.status <> ERR_FUB_BUSY AND httpClient_0.status <> 0 THEN
				httpClientErrorStatus := httpClient_0.status;
				Step := 19;
			ELSIF TON_ReloadTimeout.Q THEN // Timout! httpClient takes too long, so abort
				Status := ERR_NO_IMAGE;
				Step := 0;
			END_IF
		19: // httpclient Error
			httpClient_0.enable	:= TRUE;
			httpClient_0.send	:= FALSE;
			httpClient_0.abort	:= TRUE;
			httpClient_0();
			IF httpClient_0.status <> ERR_FUB_BUSY THEN
				httpClient_0.abort := FALSE;
				httpClient_0();
				Status := httpClientErrorStatus;
				Step := 0;
			END_IF

		20: // Save bmp/jpg file
			DiagTime.BeginSaveBMPJPG := clock_ms() - DiagStartTime;
			FileCreate_0.enable		:= TRUE;
			FileCreate_0.pDevice	:= ADR(CFG.FileDevice);
			FileCreate_0.pFile		:= ADR(FileNameImg);
			FileCreate_0();
			IF FileCreate_0.status = ERR_OK THEN
				Step := 21;
			ELSIF FileCreate_0.status <> ERR_FUB_BUSY THEN
				Status := FileCreate_0.status;
				Step := 0;
			END_IF
		21:
			FileWrite_0.enable		:= TRUE;
			FileWrite_0.ident		:= FileCreate_0.ident;
			FileWrite_0.offset		:= 0;
			FileWrite_0.pSrc		:= MemInfo.UploadAdr;
			FileWrite_0.len			:= UploadedImgSize;
			FileWrite_0();
			IF FileWrite_0.status = ERR_OK THEN
				Step := 22;
			ELSIF FileWrite_0.status <> ERR_FUB_BUSY THEN
				Status := FileWrite_0.status;
				Step := 0;
			END_IF
		22:
			FileClose_0.enable		:= TRUE;
			FileClose_0.ident		:= FileCreate_0.ident;
			FileClose_0();
			IF FileClose_0.status = ERR_OK THEN
				DiagTime.EndSaveBMPJPG := clock_ms() - DiagStartTime;
				IF CFG.UploadSVG THEN
					Step := 30;
				ELSE // ready
					Status := 0;
					Step := 0;
				END_IF
			ELSIF FileClose_0.status <> ERR_FUB_BUSY THEN
				Status := FileClose_0.status;
				Step := 0;
			END_IF

		30: // Create SVG file with image and crosshair/texts
			DiagTime.BeginSVG := clock_ms() - DiagStartTime;
			b64neededOutput	:= (UploadedImgSize/3)*4 + BOOL_TO_UDINT(UDINT_TO_BOOL(UploadedImgSize MOD 3))*4;
			IF b64neededOutput < MemInfo.SvgSize - MemInfo.SvgHeaderSize - MemInfo.CrosshSize THEN
				brsmemset(MemInfo.SvgAdr, 0, MemInfo.SvgSize); // clear complete memory
				// Prepare the svg header up to the base64 picture data
				brsstrcpy(MemInfo.SvgAdr, ADR(SvgTexts.ContentStart));
				brsstrcat(MemInfo.SvgAdr, ADR(FileNameSvg));
				brsstrcat(MemInfo.SvgAdr, ADR(SvgTexts.ContentAfterTitle));
				IF CFG.Format = 0 THEN
					brsstrcat(MemInfo.SvgAdr, ADR('jpg'));
				ELSE
					brsstrcat(MemInfo.SvgAdr, ADR('bmp'));
				END_IF
				brsstrcat(MemInfo.SvgAdr, ADR(SvgTexts.ContentBase64));
				Step := 31;
			ELSE
				Status := ERR_BUFF_SVG;
				Step := 0;
			END_IF

		31: // Code picture data with Base64 to embedd the picture into a svg file
			b64AdrInBuffer	:= MemInfo.UploadAdr; // Original bmp or jpg picture
			b64AdrOutBuffer	:= MemInfo.SvgAdr + brsstrlen(MemInfo.SvgAdr); // Write to the end of the actual svg data
			b64actposIN		:= b64AdrInBuffer;
			b64actposOUT	:= b64AdrOutBuffer;
			Step := 32;
		32: // Convert
			FOR i := 0 TO CFG.ConvertCycles DO
				IF b64actposIN < b64AdrInBuffer + UploadedImgSize THEN
					b64blockLen := UDINT_TO_USINT(LIMIT(0, b64AdrInBuffer + UploadedImgSize - b64actposIN, 3));
					b64in ACCESS b64actposIN;
					b64out ACCESS b64actposOUT;
					b64out[0]		:= b64key[ SHR(b64in[0],2) ];	// always
					IF b64blockLen = 1 THEN
						b64out[1]	:= b64key[ SHL((b64in[0] AND 16#03),4)];
						b64out[2]	:= 61;	// 61 = '='
						b64out[3]	:= 61;	// 61 = '='
					ELSIF b64blockLen = 2 THEN
						b64out[1]	:= b64key[ SHL((b64in[0] AND 16#03),4) OR SHR(b64in[1],4) ];
						b64out[2]	:= b64key[ SHL((b64in[1] AND 16#0F),2)];
						b64out[3]	:= 61;	// 61 = '='
					ELSIF b64blockLen = 3 THEN
						b64out[1]	:= b64key[ SHL((b64in[0] AND 16#03),4) OR SHR(b64in[1],4) ];
						b64out[2]	:= b64key[ SHL((b64in[1] AND 16#0F),2) OR SHR(b64in[2],6) ];
						b64out[3]	:= b64key[ b64in[2] AND 16#3F ];
					END_IF
					b64actposIN		:= b64actposIN + 3;
					b64actposOUT	:= b64actposOUT + 4;
				ELSE
					Step := 33;
					EXIT;
				END_IF
			END_FOR

		33: // Prepare the second part after base64 picture data
			brsmemset(MemInfo.CrosshAdr, 0, MemInfo.CrosshSize);
			brsstrcat(MemInfo.CrosshAdr, ADR(SvgTexts.ContentBeginJS));
			brsstrcat(MemInfo.CrosshAdr, ADR(CrossHairInfo[1].DataVis));
			brsstrcat(MemInfo.CrosshAdr, ADR(SvgTexts.ContentBetween1));
			FirstElement := TRUE;
			FOR i := 1 TO MAX_NUM_RESULTS DO
				IF CrossHairInfo[i].CrosshairTopLeftX <> 0 AND CrossHairInfo[i].CrosshairTopLeftY <> 0 THEN
					IF FirstElement THEN
						FirstElement := FALSE;
					ELSE
						brsstrcat(MemInfo.CrosshAdr, ADR(SvgTexts.ContentBetween2)); // Needed between the elements
					END_IF
					brsstrcat(MemInfo.CrosshAdr, ADR(CrossHairInfo[i].Data));
				END_IF
			END_FOR
			brsstrcat(MemInfo.CrosshAdr, ADR(SvgTexts.ContentEndJS));

			// Create the crosshairs
			FOR i := 1 TO MAX_NUM_RESULTS DO
				IF CrossHairInfo[i].CrosshairTopLeftX <> 0 AND CrossHairInfo[i].CrosshairTopLeftY <> 0 THEN
					brsstrcat(MemInfo.CrosshAdr, ADR(SvgTexts.ContentCrossHairBegin));
					brsitoa(i, ADR(tmpStr1));
					brsstrcat(MemInfo.CrosshAdr, ADR(tmpStr1));
					brsstrcat(MemInfo.CrosshAdr, ADR(SvgTexts.ContentCrossHairMiddle));
					brsitoa(REAL_TO_DINT(CrossHairInfo[i].CrosshairTopLeftX), ADR(tmpStr1));
					brsstrcat(MemInfo.CrosshAdr, ADR(tmpStr1));
					brsstrcat(MemInfo.CrosshAdr, ADR(','));
					brsitoa(REAL_TO_DINT(CrossHairInfo[i].CrosshairTopLeftY), ADR(tmpStr1));
					brsstrcat(MemInfo.CrosshAdr, ADR(tmpStr1));
					brsstrcat(MemInfo.CrosshAdr, ADR(') rotate('));
					brsitoa(REAL_TO_DINT(CrossHairInfo[i].CrosshairRotateCenter), ADR(tmpStr1));
					brsstrcat(MemInfo.CrosshAdr, ADR(tmpStr1));
					brsstrcat(MemInfo.CrosshAdr, ADR(','));
					brsitoa(REAL_TO_DINT(CrossHairInfo[i].CrosshairSizeScaled / 2), ADR(tmpStr1));
					brsstrcat(MemInfo.CrosshAdr, ADR(tmpStr1));
					brsstrcat(MemInfo.CrosshAdr, ADR(','));
					brsstrcat(MemInfo.CrosshAdr, ADR(tmpStr1));
					brsstrcat(MemInfo.CrosshAdr, ADR(') scale('));
					brsitoa(REAL_TO_DINT(CrossHairInfo[i].CrosshairScale), ADR(tmpStr1));
					brsstrcat(MemInfo.CrosshAdr, ADR(tmpStr1));
					brsstrcat(MemInfo.CrosshAdr, ADR(','));
					brsstrcat(MemInfo.CrosshAdr, ADR(tmpStr1));
					brsstrcat(MemInfo.CrosshAdr, ADR(SvgTexts.ContentCrossHairEnd));
				END_IF
			END_FOR
			brsstrcat(MemInfo.CrosshAdr, ADR(SvgTexts.ContentCrossHairRed));
			// Create the indices
			FOR i := 1 TO MAX_NUM_RESULTS DO
				IF CrossHairInfo[i].CrosshairTopLeftX <> 0 AND CrossHairInfo[i].CrosshairTopLeftY <> 0 THEN
					brsstrcat(MemInfo.CrosshAdr, ADR(SvgTexts.ContentCrossHairIndex));
				END_IF
			END_FOR
			brsstrcat(MemInfo.CrosshAdr, ADR(SvgTexts.ContentEnd));
			Step := 41;
		41:
			brsstrcat(MemInfo.SvgAdr, MemInfo.CrosshAdr);
			Step := 50;
		50:
			DiagTime.BeginSVGSave := clock_ms() - DiagStartTime;
			FileCreate_0.enable		:= TRUE;
			FileCreate_0.pDevice	:= ADR(CFG.FileDevice);
			FileCreate_0.pFile		:= ADR(FileNameSvg);
			FileCreate_0();
			IF FileCreate_0.status = ERR_OK THEN
				Step := 51;
			ELSIF FileCreate_0.status <> ERR_FUB_BUSY THEN
				Status := FileCreate_0.status;
				Step := 0;
			END_IF
		51:
			FileWrite_0.enable		:= TRUE;
			FileWrite_0.ident		:= FileCreate_0.ident;
			FileWrite_0.offset		:= 0;
			FileWrite_0.pSrc		:= MemInfo.SvgAdr;
			FileWrite_0.len			:= brsstrlen(MemInfo.SvgAdr);
			FileWrite_0();
			IF FileWrite_0.status = ERR_OK THEN
				Step := 52;
			ELSIF FileWrite_0.status <> ERR_FUB_BUSY THEN
				Status := FileWrite_0.status;
				Step := 0;
			END_IF
		52:
			FileClose_0.enable		:= TRUE;
			FileClose_0.ident		:= FileCreate_0.ident;
			FileClose_0();
			IF FileClose_0.status = ERR_OK THEN
				DiagTime.EndSVGSave := clock_ms() - DiagStartTime;
				Status := 0;
				Step := 0;
			ELSIF FileClose_0.status <> ERR_FUB_BUSY THEN
				Status := FileClose_0.status;
				Step := 0;
			END_IF
	END_CASE
END_FUNCTION_BLOCK
```

#### ViShowImgOnVC4.st - not listed in the package file held
```iecst
// Note: This FBK needs to be called at least once in the INIT of the task to alloc memory (restriction of AsMem)
FUNCTION_BLOCK ViShowImgOnVC4
	IF MemInfo.UploadBmp8Adr = 0 THEN // This will only be done once in the INIT of the task
		// Create memory for uploading and transforming image
		// Size: a 5MP picture in bmp format has less than 6.000.000 Bytes. A SVG with bas64 conversion maximum the 4/3 size.
		MemInfo.UploadBmp8Size		:= 6000000;		// Upload of the picture data with httpClient
		MemInfo.Bmp24Size			:= 18000000; 	// The 24bit img could be 3 times bigger
		AsMemPartCreate_0.enable	:= TRUE;
		AsMemPartCreate_0.len		:= MemInfo.UploadBmp8Size + MemInfo.Bmp24Size + 1000; // 1000 Bytes for AsMemPart stuff/header
		AsMemPartCreate_0();
		IF AsMemPartCreate_0.status = ERR_OK THEN
			// Upload mem for loading the image from camera to plc
			AsMemPartAllocClear_0.len		:= MemInfo.UploadBmp8Size;
			AsMemPartAllocClear_0(enable := TRUE, ident := AsMemPartCreate_0.ident);
			IF AsMemPartAllocClear_0.status = ERR_OK THEN
				MemInfo.UploadBmp8Adr		:= AsMemPartAllocClear_0.mem;
			END_IF
			// Bmp24 mem for creating the new image
			AsMemPartAllocClear_0.len		:= MemInfo.Bmp24Size;
			AsMemPartAllocClear_0(enable := TRUE, ident := AsMemPartCreate_0.ident);
			IF AsMemPartAllocClear_0.status = ERR_OK THEN
				MemInfo.Bmp24Adr 			:= AsMemPartAllocClear_0.mem;
			END_IF
		END_IF
	END_IF
	IF NOT Enable THEN
		HTMLStreamContent	:= '<p>Ready</p>';
		RefreshDone			:= FALSE;
		Status := ERR_FUB_ENABLE_FALSE;
		Step := 0;
		RETURN;
	END_IF
	CASE Step OF
		0:
			RefreshDone := FALSE;
			Status := ERR_FUB_BUSY;
			IF MemInfo.UploadBmp8Adr <> 0 AND MemInfo.Bmp24Adr <> 0 THEN
				IF RefreshImage THEN
					Step := 1;
				END_IF
			END_IF
		1: // Initialization
			CreateVC4HTML;
			FileNameBmp24Bit	:= 'http://localhost/CamImgVC4.bmp';
			FileNameBmp24BitDir	:= 'web/CamImgVC4.bmp';
			// Create URI and Host
			URI := '/bmp';
			Host := CFG.PlkIPWithoutNode;
			brsitoa(PowerlinkNode, ADR(tmpStr1));
			brsstrcat(ADR(Host), ADR(tmpStr1));
			HTMLStreamContent := '<p>Please wait... image will be loaded...</p>';
			Step := 10;
		10: // Reset timer and HTTP client
			TON_Timeout(IN := FALSE);
			httpClient_0(enable := FALSE, abort := FALSE, send := FALSE);
			IF httpClient_0.status = ERR_FUB_ENABLE_FALSE THEN
				Step := 11;
			END_IF

		11: // Wait for response
			TON_Timeout(IN := TRUE, PT := T#10s); // Time out when no response after 10s
			RequestHeader.keepAlive			:= 'timeout=5, max=100';
			httpClient_0.enable				:= TRUE;
			httpClient_0.send				:= TRUE;
			httpClient_0.method 			:= httpMETHOD_GET;
			httpClient_0.option 			:= httpOPTION_HTTP_11;
			httpClient_0.hostPort			:= 8080;
			httpClient_0.pHost 				:= ADR(Host);
			httpClient_0.pUri 				:= ADR(URI);
			httpClient_0.pResponseData 		:= MemInfo.UploadBmp8Adr;
			httpClient_0.responseDataSize	:= MemInfo.UploadBmp8Size;
			httpClient_0.pRequestHeader		:= ADR(RequestHeader);
			httpClient_0();
			IF httpClient_0.status = ERR_OK AND httpClient_0.responseDataLen <> 0 THEN
				FileSizeIn8Bit				:= httpClient_0.responseDataLen;
				httpClient_0(send := FALSE);
				IF FileSizeIn8Bit < 100 THEN // No image available. Hint: In case of no image there will be sent 86 Bytes with an html error text
					HTMLStreamContent := '<p>No image found on the camera</p>';
					Status := ERR_NO_IMAGE;
					Step := 50;
				ELSE
					Step := 20;
				END_IF
			ELSIF httpClient_0.status <> ERR_FUB_BUSY AND httpClient_0.status <> 0 THEN
				httpClientErrorStatus := httpClient_0.status;
				Step := 19;
			ELSIF TON_Timeout.Q THEN // Timout! httpClient takes too long, so abort
				HTMLStreamContent := '<p>Timeout while loading image</p>';
				Status := ERR_NO_IMAGE;
				Step := 50;
			END_IF
		19: // httpclient Error
			httpClient_0.enable	:= TRUE;
			httpClient_0.send	:= FALSE;
			httpClient_0.abort	:= TRUE;
			httpClient_0();
			IF httpClient_0.status <> ERR_FUB_BUSY THEN
				httpClient_0.abort := FALSE;
				httpClient_0();
				Status := httpClientErrorStatus;
				Step := 50;
			END_IF

		20: // Convert image from 8 bit bmp with color table to 24 bit bmp image
			brsmemcpy(ADR(Bmp8Bit)+2, MemInfo.UploadBmp8Adr, SIZEOF(Bmp8Bit)); // Use the read data
			brsmemcpy(ADR(Bmp24Bit), ADR(Bmp8Bit), SIZEOF(Bmp24Bit)); // Copy the header, but not the colour data
			// Change and add fileheader
			Bmp24Bit.InfoHeader.biBitCount	:= 24;
			Bmp24Bit.FileHeader.bfOffBits	:= SIZEOF(Bmp24Bit)-2;
			brsmemcpy(MemInfo.Bmp24Adr, ADR(Bmp24Bit)+2, SIZEOF(Bmp24Bit)-2);
			// Generate pixels
			BytesPerLine := Bmp24Bit.InfoHeader.biWidth;
			IF BytesPerLine MOD 4 > 0 THEN // Add fill bytes if necessary. The lengt of a line is always a multiple of 4.
				BytesPerLine := BytesPerLine + (4 - BytesPerLine MOD 4);
			END_IF
			IF Bmp8Bit.FileHeader.bfOffBits > (14+40+4*255) AND BytesPerLine > 0 AND ABS(Bmp24Bit.InfoHeader.biHeight) > 0 THEN // Header 14+40 + ColorTable
				PixelSourceAdr	:= MemInfo.UploadBmp8Adr + Bmp8Bit.FileHeader.bfOffBits;
				PixelDestAdr	:= MemInfo.Bmp24Adr + SIZEOF(Bmp24Bit)-2; // directly start after the header. -2 because of two fillbyts at the beginning
				BytesRemaining	:= BytesPerLine * ABS(Bmp24Bit.InfoHeader.biHeight);
				Step := 21;
			ELSE
				Status := ERR_DATA_BMP;
				Step := 50;
			END_IF
		21:
			FOR i := 0 TO CFG.ConvertCycles DO
				PixelSourceColor ACCESS PixelSourceAdr;
				PixelDestColor ACCESS PixelDestAdr;
				PixelDestColor.Blue		:= Bmp8Bit.ColorTable[PixelSourceColor].Blue;
				PixelDestColor.Green	:= Bmp8Bit.ColorTable[PixelSourceColor].Green;
				PixelDestColor.Red		:= Bmp8Bit.ColorTable[PixelSourceColor].Red;
				BytesRemaining := BytesRemaining - 1;
				IF BytesRemaining = 0 THEN
					Step := 30;
					EXIT;
				ELSE
					PixelSourceAdr		:= PixelSourceAdr + 1;
					PixelDestAdr		:= PixelDestAdr + 3;
					IF PixelSourceAdr > MemInfo.UploadBmp8Adr + MemInfo.UploadBmp8Size - 1 OR PixelDestAdr + 2 > MemInfo.Bmp24Adr + MemInfo.Bmp24Size -1 THEN
						Status := ERR_BUFF_BMP;
						Step := 50;
						EXIT;
					END_IF
				END_IF
			END_FOR

		30: // Save content to a bmp file
			FileDelete_0.enable		:= TRUE;
			FileDelete_0.pDevice	:= ADR(CFG.FileDevice);
			FileDelete_0.pName		:= ADR(FileNameBmp24BitDir);
			FileDelete_0();
			IF FileDelete_0.status = ERR_OK OR FileDelete_0.status = fiERR_FILE_NOT_FOUND THEN
				Step := 31;
			ELSIF FileDelete_0.status <> ERR_FUB_BUSY THEN
				Status := FileDelete_0.status;
				Step := 100;
			END_IF
		31:
			FileCreate_0.enable		:= TRUE;
			FileCreate_0.pDevice	:= ADR(CFG.FileDevice);
			FileCreate_0.pFile		:= ADR(FileNameBmp24BitDir);
			FileCreate_0();
			IF FileCreate_0.status = ERR_OK THEN
				Step := 32;
			ELSIF FileCreate_0.status <> ERR_FUB_BUSY THEN
				Status := FileCreate_0.status;
				Step := 100;
			END_IF
		32:
			FileWrite_0.enable		:= TRUE;
			FileWrite_0.ident		:= FileCreate_0.ident;
			FileWrite_0.pSrc		:= MemInfo.Bmp24Adr;
			FileWrite_0.len			:= MIN(MemInfo.Bmp24Size, PixelDestAdr - MemInfo.Bmp24Adr);
			FileWrite_0();
			IF FileWrite_0.status = ERR_OK THEN
				Step := 33;
			ELSIF FileWrite_0.status <> ERR_FUB_BUSY THEN
				Status := FileWrite_0.status;
				Step := 100;
			END_IF
		33:
			FileClose_0.enable	:= TRUE;
			FileClose_0.ident	:= FileCreate_0.ident;
			FileClose_0();
			IF FileClose_0.status = ERR_OK THEN
				Step := 40;
			ELSIF FileClose_0.status <> ERR_FUB_BUSY THEN
				Status := FileClose_0.status;
				Step := 100;
			END_IF

		40: // Create content for VC4 html control element
			ImgHeight_px := UDINT_TO_UINT(UINT_TO_UDINT(ImgWidthInVC4_px) *1024 / 1280);
			brsstrcpy(ADR(HTMLStreamContent), ADR(VC4HTML[0]));
			brsitoa(ImgWidthInVC4_px, ADR(tmpStr1));
			brsstrcat(ADR(HTMLStreamContent), ADR(tmpStr1));
			brsstrcat(ADR(HTMLStreamContent), ADR(VC4HTML[1]));
			brsitoa(ImgHeight_px, ADR(tmpStr1));
			brsstrcat(ADR(HTMLStreamContent), ADR(tmpStr1));
			brsstrcat(ADR(HTMLStreamContent), ADR(VC4HTML[2]));
			brsstrcat(ADR(HTMLStreamContent), ADR(FileNameBmp24Bit));
			brsstrcat(ADR(HTMLStreamContent), ADR(VC4HTML[3]));
			Status := 0;
			Step := 50;

		50:
			RefreshDone := TRUE;
			IF NOT RefreshImage THEN
				RefreshDone := FALSE;
				Step := 0;
			END_IF
	END_CASE
END_FUNCTION_BLOCK
```

### Program Logical/Vision/Vi_nettime (IEC)

#### Variables.var
```iecst
VAR
	PowerlinkCycle_us : DINT; (*Powerlink cycletime in microseconds*)
	NettimeLastCycle_us : DINT; (*Old nettime used to calculate Powerlink cycle time*)
	AxisPositionNow : LREAL; (*Calculated positon of the axis position, acopos and network delay times are compensated*)
	TriggerTimeDelta_us : DINT; (*Delta time in microseconds to the next trigger*)
	TriggerPosDelta : LREAL; (*Delta position in units to the next trigger*)
END_VAR
```
